C05493=1117.281,-65.338,-48.036,179.657,5.180,148.998
C05494=1117.275,-65.089,-48.047,179.658,5.185,148.999
C05495=1117.270,-64.839,-48.058,179.658,5.190,149.000
C05496=1117.264,-64.590,-48.069,179.659,5.196,149.001
C05497=1117.259,-64.339,-48.080,179.659,5.201,149.001
C05498=1117.254,-64.090,-48.090,179.659,5.206,149.003
C05499=1117.249,-63.840,-48.101,179.660,5.211,149.004
C05500=1117.244,-63.590,-48.112,179.660,5.216,149.004
C05501=1117.239,-63.341,-48.123,179.661,5.222,149.005
C05502=1117.233,-63.091,-48.134,179.661,5.227,149.007
C05503=1117.228,-62.842,-48.145,179.661,5.231,149.007
C05504=1117.223,-62.592,-48.156,179.662,5.237,149.008
C05505=1117.217,-62.342,-48.166,179.663,5.242,149.009
C05506=1117.212,-62.093,-48.178,179.664,5.247,149.010
C05507=1117.207,-61.842,-48.189,179.664,5.252,149.011
C05508=1117.202,-61.593,-48.200,179.665,5.258,149.012
C05509=1117.197,-61.343,-48.210,179.665,5.263,149.013
C05510=1117.191,-61.093,-48.222,179.665,5.268,149.014
C05511=1117.186,-60.844,-48.233,179.666,5.273,149.015
C05512=1117.181,-60.594,-48.244,179.667,5.278,149.016
C05513=1117.176,-60.344,-48.255,179.668,5.283,149.017
C05514=1117.170,-60.094,-48.266,179.668,5.288,149.018
C05515=1117.166,-59.880,-48.276,179.668,5.292,149.019
C05516=1117.161,-59.664,-48.285,179.668,5.296,149.020
C05517=1117.157,-59.450,-48.294,179.668,5.301,149.021
C05518=1117.153,-59.235,-48.304,179.668,5.305,149.022
C05519=1117.148,-59.020,-48.313,179.668,5.309,149.022
C05520=1117.143,-58.805,-48.323,179.668,5.313,149.023
C05521=1117.139,-58.590,-48.333,179.667,5.317,149.024
C05522=1117.134,-58.375,-48.343,179.667,5.321,149.025
C05523=1117.129,-58.124,-48.353,179.668,5.325,149.026
C05524=1117.123,-57.875,-48.365,179.667,5.330,149.027
C05525=1117.119,-57.626,-48.376,179.667,5.335,149.028
C05526=1117.114,-57.376,-48.387,179.667,5.339,149.029
C05527=1117.108,-57.126,-48.398,179.666,5.344,149.031
C05528=1117.103,-56.877,-48.409,179.666,5.349,149.032
C05529=1117.098,-56.627,-48.421,179.666,5.353,149.033
C05530=1117.093,-56.377,-48.433,179.666,5.358,149.034
C05531=1117.087,-56.127,-48.443,179.666,5.362,149.035
C05532=1117.082,-55.877,-48.455,179.666,5.367,149.036
C05533=1117.077,-55.628,-48.466,179.666,5.372,149.037
C05534=1117.072,-55.379,-48.477,179.666,5.376,149.038
C05535=1117.066,-55.128,-48.488,179.665,5.381,149.039
C05536=1117.061,-54.879,-48.499,179.665,5.386,149.040
C05537=1117.056,-54.629,-48.511,179.665,5.391,149.041
C05538=1117.051,-54.380,-48.522,179.665,5.396,149.042
C05539=1117.046,-54.130,-48.533,179.664,5.400,149.043
C05540=1117.040,-53.880,-48.545,179.665,5.405,149.044
C05541=1117.036,-53.630,-48.556,179.664,5.409,149.045
C05542=1117.029,-53.381,-48.567,179.664,5.414,149.047
C05543=1117.025,-53.131,-48.579,179.664,5.419,149.048
C05544=1117.019,-52.881,-48.591,179.664,5.423,149.049
C05545=1117.015,-52.632,-48.602,179.664,5.429,149.050
C05546=1117.009,-52.382,-48.613,179.663,5.432,149.051
C05547=1117.004,-52.132,-48.624,179.663,5.438,149.052
C05548=1116.998,-51.882,-48.636,179.663,5.443,149.053
C05549=1116.994,-51.633,-48.647,179.663,5.447,149.054
C05550=1116.987,-51.383,-48.659,179.663,5.452,149.055
C05551=1116.983,-51.134,-48.670,179.662,5.456,149.056
C05552=1116.977,-50.884,-48.682,179.663,5.461,149.057
C05553=1116.973,-50.634,-48.693,179.663,5.466,149.058
C05554=1116.967,-50.384,-48.705,179.662,5.470,149.060
C05555=1116.962,-50.135,-48.716,179.662,5.476,149.061
C05556=1116.957,-49.885,-48.728,179.662,5.479,149.062
C05557=1116.952,-49.636,-48.739,179.662,5.485,149.063
C05558=1116.946,-49.385,-48.750,179.662,5.490,149.064
C05559=1116.941,-49.136,-48.762,179.661,5.494,149.065
C05560=1116.935,-48.886,-48.773,179.661,5.499,149.066
C05561=1116.931,-48.637,-48.784,179.661,5.503,149.067
C05562=1116.925,-48.387,-48.796,179.661,5.508,149.068
C05563=1116.920,-48.137,-48.808,179.661,5.513,149.069
C05564=1116.915,-47.887,-48.819,179.660,5.517,149.070
C05565=1116.909,-47.638,-48.831,179.660,5.522,149.071
C05566=1116.904,-47.388,-48.842,179.660,5.526,149.072
C05567=1116.899,-47.138,-48.854,179.660,5.532,149.073
C05568=1116.894,-46.889,-48.865,179.660,5.537,149.075
C05569=1116.889,-46.639,-48.877,179.659,5.541,149.076
C05570=1116.884,-46.390,-48.890,179.660,5.546,149.077
C05571=1116.879,-46.174,-48.899,179.660,5.550,149.078
C05572=1116.875,-45.959,-48.909,179.659,5.554,149.079
C05573=1116.870,-45.744,-48.919,179.659,5.558,149.079
C05574=1116.866,-45.529,-48.929,179.659,5.562,149.081
C05575=1116.862,-45.315,-48.939,179.658,5.566,149.081
C05576=1116.857,-45.099,-48.950,179.658,5.570,149.082
C05577=1116.852,-44.885,-48.959,179.659,5.575,149.083
C05578=1116.847,-44.670,-48.969,179.658,5.579,149.084
C05579=1116.843,-44.421,-48.981,179.658,5.583,149.085
C05580=1116.837,-44.171,-48.993,179.658,5.588,149.086
C05581=1116.832,-43.921,-49.005,179.658,5.592,149.087
C05582=1116.827,-43.671,-49.016,179.658,5.597,149.089
C05583=1116.822,-43.422,-49.028,179.658,5.602,149.089
C05584=1116.817,-43.172,-49.040,179.657,5.606,149.091
C05585=1116.812,-42.922,-49.052,179.657,5.611,149.092
C05586=1116.806,-42.672,-49.063,179.658,5.617,149.093
C05587=1116.801,-42.422,-49.075,179.660,5.622,149.093
C05588=1116.796,-42.174,-49.086,179.661,5.628,149.094
C05589=1116.791,-41.924,-49.099,179.662,5.633,149.095
C05590=1116.785,-41.674,-49.111,179.663,5.638,149.096
C05591=1116.780,-41.424,-49.123,179.664,5.644,149.097
C05592=1116.775,-41.175,-49.134,179.665,5.649,149.098
C05593=1116.770,-40.925,-49.147,179.666,5.654,149.098
C05594=1116.765,-40.676,-49.158,179.667,5.659,149.099
C05595=1116.759,-40.426,-49.170,179.668,5.665,149.100
C05596=1116.754,-40.176,-49.182,179.669,5.669,149.101
C05597=1116.749,-39.927,-49.194,179.670,5.675,149.102
C05598=1116.744,-39.677,-49.206,179.672,5.680,149.103
C05599=1116.738,-39.427,-49.218,179.672,5.685,149.103
C05600=1116.733,-39.177,-49.231,179.673,5.690,149.104
C05601=1116.729,-38.928,-49.242,179.674,5.695,149.105
C05602=1116.723,-38.678,-49.254,179.675,5.699,149.106
C05603=1116.718,-38.429,-49.266,179.676,5.705,149.107
C05604=1116.713,-38.179,-49.278,179.676,5.710,149.108
C05605=1116.707,-37.929,-49.290,179.677,5.714,149.108
C05606=1116.702,-37.679,-49.303,179.678,5.719,149.109
C05607=1116.697,-37.430,-49.314,179.679,5.724,149.110
C05608=1116.692,-37.180,-49.327,179.680,5.729,149.111
C05609=1116.687,-36.930,-49.339,179.680,5.733,149.112
C05610=1116.681,-36.681,-49.350,179.681,5.738,149.113
C05611=1116.676,-36.431,-49.363,179.682,5.743,149.113
C05612=1116.671,-36.181,-49.375,179.683,5.748,149.114
C05613=1116.666,-35.932,-49.387,179.683,5.753,149.115
C05614=1116.660,-35.682,-49.399,179.683,5.757,149.116
C05615=1116.655,-35.433,-49.412,179.684,5.762,149.117
C05616=1116.650,-35.183,-49.423,179.685,5.766,149.117
C05617=1116.645,-34.934,-49.436,179.685,5.771,149.118
C05618=1116.640,-34.684,-49.448,179.685,5.775,149.119
C05619=1116.635,-34.435,-49.460,179.686,5.780,149.120
C05620=1116.629,-34.185,-49.472,179.687,5.784,149.121
C05621=1116.625,-33.935,-49.485,179.687,5.789,149.122
C05622=1116.619,-33.685,-49.497,179.687,5.794,149.123
C05623=1116.614,-33.435,-49.510,179.687,5.798,149.124
C05624=1116.609,-33.186,-49.522,179.688,5.802,149.124
C05625=1116.604,-32.936,-49.534,179.689,5.807,149.125
C05626=1116.599,-32.687,-49.547,179.689,5.811,149.126
C05627=1116.594,-32.472,-49.557,179.689,5.815,149.127
C05628=1116.589,-32.257,-49.568,179.689,5.819,149.128
C05629=1116.586,-32.042,-49.578,179.690,5.823,149.128
C05630=1116.581,-31.827,-49.589,179.690,5.826,149.129
C05631=1116.577,-31.612,-49.600,179.690,5.830,149.130
C05632=1116.572,-31.397,-49.610,179.690,5.834,149.131
C05633=1116.568,-31.183,-49.621,179.690,5.838,149.132
C05634=1116.562,-30.968,-49.632,179.690,5.841,149.132
C05635=1116.557,-30.718,-49.644,179.690,5.845,149.133
C05636=1116.553,-30.468,-49.657,179.690,5.850,149.134
C05637=1116.547,-30.218,-49.669,179.690,5.854,149.135
C05638=1116.542,-29.969,-49.682,179.690,5.858,149.136
C05639=1116.537,-29.720,-49.694,179.690,5.863,149.137
C05640=1116.532,-29.470,-49.706,179.690,5.867,149.138
C05641=1116.527,-29.221,-49.719,179.690,5.871,149.139
C05642=1116.522,-28.971,-49.732,179.690,5.876,149.140
C05643=1116.517,-28.721,-49.744,179.690,5.880,149.141
C05644=1116.512,-28.471,-49.756,179.689,5.884,149.142
C05645=1116.506,-28.222,-49.769,179.689,5.888,149.143
C05646=1116.501,-27.972,-49.781,179.689,5.892,149.144
C05647=1116.496,-27.723,-49.793,179.689,5.896,149.145
C05648=1116.491,-27.473,-49.806,179.689,5.901,149.146
C05649=1116.486,-27.223,-49.819,179.688,5.906,149.147
C05650=1116.480,-26.973,-49.831,179.688,5.910,149.148
C05651=1116.475,-26.724,-49.844,179.687,5.914,149.149
C05652=1116.470,-26.475,-49.857,179.687,5.918,149.150
C05653=1116.465,-26.224,-49.870,179.686,5.922,149.151
C05654=1116.460,-25.975,-49.881,179.686,5.927,149.152
C05655=1116.455,-25.725,-49.894,179.686,5.930,149.153
C05656=1116.450,-25.476,-49.907,179.686,5.936,149.154
C05657=1116.444,-25.227,-49.919,179.687,5.941,149.155
C05658=1116.440,-24.977,-49.932,179.687,5.946,149.156
C05659=1116.434,-24.726,-49.945,179.688,5.951,149.157
C05660=1116.429,-24.477,-49.957,179.688,5.955,149.158
C05661=1116.424,-24.228,-49.970,179.689,5.960,149.159
C05662=1116.418,-23.978,-49.983,179.689,5.965,149.160
C05663=1116.414,-23.728,-49.996,179.690,5.969,149.160
C05664=1116.409,-23.479,-50.008,179.691,5.974,149.161
C05665=1116.403,-23.229,-50.021,179.692,5.979,149.162
C05666=1116.397,-22.979,-50.033,179.692,5.984,149.163
C05667=1116.393,-22.729,-50.046,179.693,5.989,149.164
C05668=1116.388,-22.480,-50.059,179.693,5.994,149.165
C05669=1116.383,-22.231,-50.071,179.694,5.998,149.166
C05670=1116.377,-21.981,-50.085,179.694,6.003,149.167
C05671=1116.372,-21.731,-50.098,179.694,6.008,149.168
C05672=1116.367,-21.482,-50.110,179.695,6.013,149.169
C05673=1116.362,-21.233,-50.123,179.695,6.017,149.169
C05674=1116.357,-20.982,-50.136,179.696,6.022,149.170
C05675=1116.352,-20.733,-50.149,179.696,6.027,149.171
C05676=1116.347,-20.484,-50.161,179.697,6.031,149.172
C05677=1116.341,-20.234,-50.174,179.698,6.036,149.173
C05678=1116.336,-19.984,-50.188,179.698,6.041,149.174
C05679=1116.331,-19.735,-50.200,179.699,6.045,149.175
C05680=1116.326,-19.485,-50.213,179.699,6.050,149.175
C05681=1116.321,-19.235,-50.226,179.700,6.055,149.176
C05682=1116.316,-18.986,-50.239,179.701,6.060,149.177
C05683=1116.311,-18.771,-50.250,179.701,6.064,149.178
C05684=1116.307,-18.556,-50.261,179.702,6.067,149.179
C05685=1116.302,-18.341,-50.272,179.702,6.072,149.179
C05686=1116.297,-18.126,-50.283,179.702,6.076,149.180
C05687=1116.293,-17.912,-50.294,179.703,6.080,149.181
C05688=1116.289,-17.697,-50.306,179.704,6.084,149.181
C05689=1116.284,-17.482,-50.317,179.704,6.088,149.182
C05690=1116.280,-17.268,-50.328,179.705,6.092,149.183
C05691=1116.275,-17.018,-50.341,179.705,6.097,149.184
C05692=1116.270,-16.768,-50.354,179.706,6.101,149.185
C05693=1116.265,-16.518,-50.367,179.707,6.106,149.186
C05694=1116.260,-16.269,-50.380,179.707,6.110,149.186
C05695=1116.254,-16.020,-50.394,179.708,6.115,149.187
C05696=1116.250,-15.770,-50.407,179.708,6.120,149.188
C05697=1116.244,-15.520,-50.420,179.709,6.124,149.189
C05698=1116.239,-15.271,-50.433,179.710,6.129,149.190
C05699=1116.234,-15.021,-50.446,179.710,6.134,149.191
C05700=1116.228,-14.771,-50.459,179.711,6.138,149.192
C05701=1116.224,-14.522,-50.473,179.711,6.143,149.192
C05702=1116.219,-14.272,-50.485,179.712,6.147,149.193
C05703=1116.213,-14.023,-50.498,179.713,6.152,149.194
C05704=1116.209,-13.773,-50.511,179.713,6.157,149.195
C05705=1116.203,-13.524,-50.525,179.714,6.162,149.196
C05706=1116.198,-13.274,-50.538,179.715,6.166,149.196
C05707=1116.193,-13.024,-50.551,179.715,6.171,149.197
C05708=1116.188,-12.774,-50.564,179.716,6.175,149.198
C05709=1116.183,-12.525,-50.578,179.716,6.180,149.199
C05710=1116.178,-12.275,-50.591,179.717,6.184,149.200
C05711=1116.172,-12.025,-50.604,179.718,6.189,149.201
C05712=1116.167,-11.777,-50.618,179.718,6.194,149.202
C05713=1116.162,-11.526,-50.631,179.719,6.199,149.202
C05714=1116.157,-11.277,-50.644,179.719,6.202,149.203
C05715=1116.152,-11.027,-50.658,179.719,6.207,149.204
C05716=1116.147,-10.778,-50.671,179.720,6.212,149.205
C05717=1116.142,-10.528,-50.684,179.721,6.216,149.206
C05718=1116.137,-10.279,-50.698,179.721,6.221,149.206
C05719=1116.131,-10.029,-50.711,179.722,6.225,149.207
C05720=1116.127,-9.780,-50.725,179.722,6.230,149.208
C05721=1116.121,-9.530,-50.738,179.723,6.234,149.209
C05722=1116.116,-9.280,-50.751,179.724,6.239,149.210
C05723=1116.111,-9.031,-50.765,179.724,6.244,149.211
C05724=1116.106,-8.781,-50.778,179.725,6.248,149.211
C05725=1116.101,-8.532,-50.792,179.726,6.253,149.212
C05726=1116.095,-8.282,-50.805,179.726,6.258,149.213
C05727=1116.091,-8.033,-50.819,179.727,6.262,149.214
C05728=1116.085,-7.783,-50.832,179.727,6.266,149.215
C05729=1116.081,-7.534,-50.846,179.728,6.271,149.216
C05730=1116.075,-7.284,-50.859,179.728,6.275,149.216
C05731=1116.070,-7.034,-50.873,179.729,6.280,149.217
C05732=1116.066,-6.784,-50.886,179.730,6.284,149.218
C05733=1116.060,-6.535,-50.900,179.730,6.289,149.219
C05734=1116.055,-6.285,-50.914,179.731,6.293,149.220
C05735=1116.050,-6.036,-50.927,179.732,6.298,149.220
C05736=1116.045,-5.786,-50.940,179.732,6.303,149.221
C05737=1116.039,-5.537,-50.954,179.733,6.308,149.222
C05738=1116.035,-5.287,-50.967,179.733,6.311,149.223
C05739=1116.030,-5.073,-50.979,179.734,6.316,149.224
C05740=1116.026,-4.858,-50.991,179.734,6.319,149.224
C05741=1116.021,-4.643,-51.002,179.735,6.324,149.225
C05742=1116.018,-4.428,-51.015,179.736,6.327,149.226
C05743=1116.013,-4.214,-51.026,179.736,6.331,149.226
C05744=1116.009,-3.999,-51.038,179.737,6.335,149.227
C05745=1116.004,-3.785,-51.050,179.737,6.339,149.228
C05746=1116.000,-3.569,-51.061,179.737,6.343,149.229
C05747=1115.994,-3.320,-51.075,179.738,6.347,149.229
C05748=1115.989,-3.070,-51.089,179.739,6.352,149.230
C05749=1115.984,-2.820,-51.103,179.739,6.356,149.231
C05750=1115.979,-2.572,-51.117,179.740,6.361,149.232
C05751=1115.974,-2.321,-51.130,179.741,6.365,149.233
C05752=1115.969,-2.072,-51.144,179.741,6.370,149.234
C05753=1115.964,-1.823,-51.158,179.742,6.375,149.234
C05754=1115.959,-1.573,-51.171,179.742,6.378,149.235
C05755=1115.954,-1.324,-51.185,179.743,6.383,149.236
C05756=1115.949,-1.074,-51.199,179.743,6.388,149.237
C05757=1115.944,-0.824,-51.214,179.744,6.393,149.238
C05758=1115.938,-0.575,-51.226,179.745,6.397,149.238
C05759=1115.934,-0.325,-51.241,179.745,6.402,149.239
C05760=1115.929,-0.075,-51.255,179.746,6.406,149.240
C05761=1115.923,0.174,-51.269,179.747,6.411,149.241
C05762=1115.918,0.424,-51.282,179.747,6.415,149.242
C05763=1115.913,0.674,-51.297,179.747,6.419,149.243
C05764=1115.908,0.922,-51.310,179.748,6.424,149.244
C05765=1115.903,1.172,-51.324,179.749,6.428,149.244
C05766=1115.898,1.422,-51.338,179.749,6.433,149.245
C05767=1115.892,1.671,-51.352,179.750,6.438,149.246
C05768=1115.887,1.921,-51.366,179.751,6.443,149.247
C05769=1115.882,2.171,-51.380,179.752,6.447,149.248
C05770=1115.878,2.420,-51.394,179.752,6.452,149.248
C05771=1115.873,2.669,-51.408,179.752,6.456,149.249
C05772=1115.868,2.919,-51.422,179.753,6.460,149.250
C05773=1115.863,3.169,-51.436,179.754,6.465,149.251
C05774=1115.857,3.418,-51.450,179.754,6.469,149.252
C05775=1115.852,3.668,-51.464,179.755,6.474,149.253
C05776=1115.847,3.918,-51.478,179.755,6.479,149.254
C05777=1115.842,4.167,-51.492,179.756,6.483,149.254
C05778=1115.836,4.416,-51.506,179.757,6.488,149.255
C05779=1115.831,4.666,-51.521,179.757,6.492,149.256
C05780=1115.826,4.916,-51.535,179.757,6.496,149.257
C05781=1115.822,5.165,-51.549,179.758,6.501,149.258
C05782=1115.817,5.414,-51.562,179.758,6.506,149.259
C05783=1115.812,5.664,-51.577,179.759,6.510,149.259
C05784=1115.807,5.914,-51.591,179.760,6.515,149.260
C05785=1115.802,6.163,-51.605,179.760,6.520,149.261
C05786=1115.797,6.413,-51.620,179.761,6.524,149.262
C05787=1115.791,6.662,-51.634,179.761,6.529,149.263
C05788=1115.786,6.912,-51.648,179.762,6.534,149.264
C05789=1115.781,7.161,-51.662,179.762,6.537,149.264
C05790=1115.776,7.411,-51.676,179.763,6.542,149.265
C05791=1115.771,7.660,-51.690,179.763,6.547,149.266
C05792=1115.766,7.910,-51.705,179.764,6.551,149.267
C05793=1115.761,8.160,-51.719,179.765,6.556,149.268
C05794=1115.756,8.409,-51.733,179.765,6.561,149.269
C05795=1115.750,8.699,-51.750,179.766,6.566,149.270
C05796=1115.744,8.990,-51.767,179.766,6.571,149.271
C05797=1115.737,9.281,-51.783,179.767,6.577,149.272
C05798=1115.732,9.572,-51.800,179.768,6.582,149.273
C05799=1115.727,9.822,-51.815,179.769,6.586,149.273
C05800=1115.722,10.072,-51.829,179.769,6.591,149.274
C05801=1115.717,10.320,-51.844,179.770,6.596,149.275
C05802=1115.712,10.570,-51.858,179.770,6.600,149.276
C05803=1115.707,10.819,-51.872,179.771,6.605,149.277
C05804=1115.702,11.069,-51.886,179.772,6.610,149.278
C05805=1115.697,11.319,-51.901,179.772,6.614,149.278
C05806=1115.692,11.568,-51.916,179.773,6.619,149.279
C05807=1115.687,11.818,-51.931,179.774,6.623,149.280
C05808=1115.681,12.067,-51.944,179.774,6.628,149.281
C05809=1115.676,12.317,-51.959,179.775,6.633,149.282
C05810=1115.671,12.566,-51.973,179.776,6.637,149.282
C05811=1115.667,12.816,-51.988,179.777,6.642,149.283
C05812=1115.662,13.065,-52.002,179.777,6.646,149.284
C05813=1115.657,13.315,-52.017,179.778,6.650,149.285
C05814=1115.651,13.564,-52.032,179.778,6.655,149.286
C05815=1115.646,13.814,-52.046,179.779,6.659,149.287
C05816=1115.641,14.064,-52.061,179.780,6.664,149.287
C05817=1115.636,14.313,-52.075,179.780,6.668,149.288
C05818=1115.632,14.563,-52.090,179.781,6.673,149.289
C05819=1115.625,14.812,-52.104,179.782,6.677,149.290
C05820=1115.620,15.062,-52.119,179.782,6.682,149.291
C05821=1115.616,15.311,-52.134,179.783,6.686,149.291
C05822=1115.611,15.560,-52.148,179.784,6.691,149.292
C05823=1115.606,15.810,-52.162,179.785,6.695,149.293
C05824=1115.600,16.060,-52.178,179.786,6.700,149.294
C05825=1115.596,16.309,-52.192,179.786,6.705,149.295
C05826=1115.591,16.558,-52.207,179.787,6.708,149.295
C05827=1115.586,16.808,-52.221,179.787,6.713,149.296
C05828=1115.580,17.058,-52.236,179.788,6.717,149.297
C05829=1115.576,17.307,-52.251,179.789,6.722,149.298
C05830=1115.571,17.557,-52.266,179.790,6.726,149.298
C05831=1115.563,17.945,-52.289,179.791,6.734,149.300
C05832=1115.555,18.333,-52.312,179.792,6.740,149.301
C05833=1115.547,18.721,-52.335,179.793,6.747,149.302
C05834=1115.540,19.109,-52.358,179.794,6.754,149.303
C05835=1115.535,19.358,-52.373,179.795,6.758,149.304
C05836=1115.529,19.608,-52.388,179.796,6.763,149.305
C05837=1115.524,19.858,-52.402,179.797,6.767,149.305
C05838=1115.520,20.107,-52.417,179.797,6.772,149.306
C05839=1115.514,20.357,-52.432,179.798,6.776,149.307
C05840=1115.509,20.606,-52.447,179.799,6.781,149.307
C05841=1115.504,20.856,-52.462,179.800,6.785,149.308
C05842=1115.499,21.105,-52.477,179.801,6.790,149.309
C05843=1115.494,21.354,-52.492,179.801,6.794,149.310
C05844=1115.489,21.604,-52.507,179.802,6.798,149.311
C05845=1115.484,21.853,-52.522,179.803,6.802,149.311
C05846=1115.478,22.103,-52.537,179.804,6.807,149.312
C05847=1115.475,22.317,-52.550,179.804,6.810,149.313
C05848=1115.470,22.532,-52.563,179.805,6.815,149.313
C05849=1115.466,22.746,-52.575,179.806,6.818,149.314
C05850=1115.461,22.960,-52.589,179.807,6.822,149.314
C05851=1115.458,23.175,-52.601,179.808,6.826,149.315
C05852=1115.453,23.390,-52.614,179.808,6.829,149.316
C05853=1115.449,23.604,-52.628,179.809,6.834,149.316
C05854=1115.445,23.819,-52.640,179.809,6.837,149.317
C05855=1115.439,24.068,-52.656,179.810,6.841,149.318
C05856=1115.434,24.318,-52.670,179.812,6.846,149.318
C05857=1115.429,24.567,-52.686,179.812,6.850,149.319
C05858=1115.424,24.816,-52.701,179.813,6.854,149.320
C05859=1115.419,25.067,-52.715,179.814,6.858,149.321
C05860=1115.414,25.316,-52.730,179.815,6.863,149.321
C05861=1115.409,25.565,-52.746,179.815,6.867,149.322
C05862=1115.405,25.815,-52.761,179.816,6.872,149.323
C05863=1115.399,26.065,-52.776,179.817,6.876,149.323
C05864=1115.394,26.314,-52.791,179.818,6.880,149.324
C05865=1115.389,26.563,-52.807,179.819,6.885,149.325
C05866=1115.384,26.812,-52.822,179.819,6.888,149.326
C05867=1115.379,27.062,-52.837,179.820,6.893,149.326
C05868=1115.374,27.312,-52.852,179.821,6.897,149.327
C05869=1115.369,27.562,-52.868,179.823,6.901,149.328
C05870=1115.365,27.811,-52.883,179.824,6.906,149.328
C05871=1115.359,28.060,-52.898,179.824,6.910,149.329
C05872=1115.354,28.310,-52.914,179.825,6.915,149.330
C05873=1115.349,28.559,-52.929,179.826,6.918,149.330
C05874=1115.344,28.808,-52.944,179.827,6.923,149.331
C05875=1115.339,29.058,-52.959,179.828,6.927,149.332
C05876=1115.334,29.308,-52.975,179.829,6.931,149.332
C05877=1115.329,29.557,-52.990,179.829,6.936,149.333
C05878=1115.324,29.806,-53.005,179.830,6.940,149.334
C05879=1115.319,30.056,-53.021,179.832,6.945,149.335
C05880=1115.315,30.306,-53.036,179.833,6.949,149.335
C05881=1115.309,30.555,-53.052,179.833,6.952,149.336
C05882=1115.304,30.804,-53.067,179.834,6.957,149.337
C05883=1115.299,31.053,-53.082,179.835,6.961,149.337
C05884=1115.294,31.304,-53.098,179.836,6.965,149.338
C05885=1115.289,31.553,-53.114,179.837,6.970,149.338
C05886=1115.284,31.802,-53.129,179.838,6.974,149.339
C05887=1115.279,32.051,-53.144,179.839,6.978,149.340
C05888=1115.274,32.302,-53.160,179.840,6.982,149.340
C05889=1115.269,32.551,-53.175,179.840,6.986,149.341
C05890=1115.264,32.800,-53.191,179.842,6.991,149.342
C05891=1115.259,33.049,-53.207,179.843,6.995,149.343
C05892=1115.254,33.300,-53.223,179.844,6.999,149.343
C05893=1115.249,33.549,-53.238,179.845,7.004,149.344
C05894=1115.244,33.798,-53.253,179.846,7.008,149.345
C05895=1115.238,34.047,-53.269,179.846,7.011,149.345
C05896=1115.234,34.297,-53.284,179.847,7.016,149.346
C05897=1115.229,34.546,-53.300,179.848,7.020,149.347
C05898=1115.224,34.795,-53.316,179.849,7.024,149.347
C05899=1115.219,35.046,-53.332,179.850,7.029,149.348
C05900=1115.215,35.295,-53.347,179.852,7.033,149.348
C05901=1115.209,35.544,-53.363,179.853,7.037,149.349
C05902=1115.204,35.794,-53.378,179.854,7.040,149.350
C05903=1115.200,36.008,-53.392,179.855,7.045,149.350
C05904=1115.195,36.222,-53.406,179.855,7.048,149.351
C05905=1115.191,36.436,-53.419,179.856,7.051,149.351
C05906=1115.186,36.651,-53.432,179.857,7.056,149.352
C05907=1115.182,36.866,-53.446,179.858,7.059,149.352
C05908=1115.178,37.080,-53.460,179.858,7.062,149.353
C05909=1115.174,37.294,-53.473,179.860,7.066,149.353
C05910=1115.170,37.509,-53.487,179.860,7.070,149.354
C05911=1115.165,37.758,-53.502,179.861,7.074,149.355
C05912=1115.160,38.008,-53.518,179.863,7.078,149.355
C05913=1115.155,38.258,-53.534,179.863,7.082,149.356
C05914=1115.150,38.507,-53.550,179.864,7.086,149.357
C05915=1115.144,38.756,-53.566,179.866,7.090,149.357
C05916=1115.140,39.006,-53.582,179.867,7.095,149.358
C05917=1115.135,39.255,-53.597,179.868,7.099,149.358
C05918=1115.130,39.504,-53.613,179.869,7.103,149.359
C05919=1115.125,39.754,-53.629,179.870,7.107,149.360
C05920=1115.120,40.004,-53.645,179.871,7.111,149.360
C05921=1115.115,40.253,-53.661,179.872,7.115,149.361
C05922=1115.110,40.502,-53.677,179.873,7.119,149.362
C05923=1115.105,40.751,-53.693,179.874,7.123,149.362
C05924=1115.100,41.001,-53.709,179.875,7.128,149.363
C05925=1115.095,41.251,-53.725,179.876,7.132,149.363
C05926=1115.090,41.500,-53.741,179.878,7.136,149.364
C05927=1115.085,41.750,-53.757,179.878,7.140,149.365
C05928=1115.079,41.999,-53.773,179.879,7.144,149.365
C05929=1115.075,42.249,-53.789,179.880,7.148,149.366
C05930=1115.069,42.498,-53.805,179.881,7.152,149.367
C05931=1115.066,42.747,-53.821,179.883,7.156,149.367
C05932=1115.060,42.997,-53.836,179.884,7.161,149.368
C05933=1115.056,43.246,-53.853,179.884,7.164,149.368
C05934=1115.050,43.495,-53.869,179.886,7.168,149.369
C05935=1115.046,43.745,-53.885,179.887,7.172,149.369
C05936=1115.041,43.994,-53.901,179.888,7.177,149.370
C05937=1115.036,44.244,-53.918,179.889,7.181,149.371
C05938=1115.030,44.493,-53.934,179.890,7.185,149.371
C05939=1115.026,44.743,-53.951,179.892,7.189,149.372
C05940=1115.020,44.992,-53.966,179.892,7.193,149.372
C05941=1115.016,45.242,-53.983,179.893,7.197,149.373
C05942=1115.010,45.491,-53.998,179.894,7.201,149.374
C05943=1115.006,45.741,-54.015,179.896,7.205,149.374
C05944=1115.000,45.990,-54.031,179.897,7.210,149.375
C05945=1114.996,46.240,-54.047,179.898,7.214,149.375
C05946=1114.991,46.488,-54.064,179.899,7.217,149.376
C05947=1114.986,46.739,-54.080,179.900,7.221,149.376
C05948=1114.981,46.987,-54.096,179.901,7.226,149.377
C05949=1114.976,47.237,-54.112,179.902,7.230,149.378
C05950=1114.971,47.486,-54.128,179.904,7.234,149.378
C05951=1114.967,47.736,-54.145,179.905,7.238,149.379
C05952=1114.960,47.985,-54.161,179.906,7.242,149.380
C05953=1114.956,48.235,-54.178,179.907,7.246,149.380
C05954=1114.951,48.484,-54.194,179.908,7.250,149.381
C05955=1114.946,48.734,-54.210,179.909,7.254,149.381
C05956=1114.942,48.983,-54.227,179.911,7.258,149.382
C05957=1114.937,49.232,-54.243,179.912,7.262,149.382
C05958=1114.932,49.482,-54.259,179.913,7.266,149.383
C05959=1114.927,49.696,-54.274,179.914,7.270,149.383
C05960=1114.923,49.910,-54.288,179.915,7.273,149.384
C05961=1114.918,50.125,-54.301,179.916,7.277,149.384
C05962=1114.914,50.339,-54.316,179.917,7.280,149.385
C05963=1114.911,50.554,-54.330,179.918,7.283,149.385
C05964=1114.906,50.768,-54.344,179.919,7.287,149.386
C05965=1114.902,50.982,-54.358,179.920,7.290,149.386
C05966=1114.897,51.196,-54.372,179.921,7.294,149.387
C05967=1114.893,51.446,-54.389,179.922,7.298,149.387
C05968=1114.887,51.695,-54.406,179.923,7.302,149.388
C05969=1114.883,51.944,-54.422,179.925,7.306,149.388
C05970=1114.878,52.194,-54.438,179.926,7.310,149.389
C05971=1114.873,52.443,-54.455,179.927,7.314,149.389
C05972=1114.868,52.693,-54.472,179.928,7.318,149.390
C05973=1114.863,52.942,-54.489,179.929,7.322,149.391
C05974=1114.858,53.191,-54.505,179.931,7.326,149.391
C05975=1114.854,53.441,-54.522,179.932,7.330,149.392
C05976=1114.847,53.690,-54.538,179.933,7.334,149.392
C05977=1114.843,53.940,-54.554,179.934,7.339,149.393
C05978=1114.838,54.189,-54.571,179.935,7.342,149.393
C05979=1114.833,54.438,-54.588,179.936,7.346,149.394
C05980=1114.828,54.688,-54.605,179.938,7.350,149.394
C05981=1114.824,54.937,-54.621,179.939,7.354,149.395
C05982=1114.818,55.187,-54.638,179.941,7.358,149.396
C05983=1114.813,55.436,-54.655,179.942,7.362,149.396
C05984=1114.809,55.686,-54.672,179.943,7.366,149.397
C05985=1114.803,55.935,-54.688,179.944,7.370,149.397
C05986=1114.799,56.184,-54.705,179.945,7.374,149.398
C05987=1114.794,56.434,-54.722,179.946,7.378,149.398
C05988=1114.789,56.683,-54.739,179.947,7.382,149.399
C05989=1114.784,56.932,-54.755,179.949,7.386,149.399
C05990=1114.779,57.182,-54.773,179.950,7.391,149.400
C05991=1114.774,57.431,-54.789,179.952,7.394,149.401
C05992=1114.769,57.680,-54.806,179.952,7.398,149.401
C05993=1114.764,57.930,-54.823,179.954,7.402,149.402
C05994=1114.759,58.179,-54.840,179.955,7.406,149.402
C05995=1114.754,58.429,-54.857,179.956,7.410,149.403
C05996=1114.749,58.678,-54.873,179.958,7.414,149.403
C05997=1114.744,58.927,-54.891,179.959,7.418,149.404
C05998=1114.740,59.177,-54.908,179.961,7.422,149.404
C05999=1114.735,59.426,-54.924,179.961,7.426,149.405
C06000=1114.729,59.675,-54.941,179.963,7.430,149.405
C06001=1114.725,59.925,-54.958,179.964,7.434,149.406
C06002=1114.720,60.175,-54.975,179.965,7.438,149.406
C06003=1114.715,60.424,-54.992,179.966,7.442,149.407
C06004=1114.710,60.673,-55.010,179.968,7.446,149.407
C06005=1114.705,60.922,-55.026,179.969,7.450,149.408
C06006=1114.700,61.172,-55.043,179.971,7.454,149.409
C06007=1114.696,61.421,-55.060,179.972,7.457,149.409
C06008=1114.690,61.671,-55.077,179.973,7.462,149.410
C06009=1114.686,61.920,-55.095,179.974,7.466,149.410
C06010=1114.680,62.169,-55.112,179.975,7.470,149.411
C06011=1114.676,62.419,-55.128,179.977,7.474,149.411
C06012=1114.671,62.668,-55.146,179.978,7.478,149.412
C06013=1114.666,62.918,-55.164,179.980,7.482,149.412
C06014=1114.661,63.167,-55.180,179.981,7.486,149.413
C06015=1114.656,63.381,-55.195,179.982,7.489,149.413
C06016=1114.652,63.595,-55.210,179.983,7.492,149.413
C06017=1114.648,63.809,-55.225,179.985,7.496,149.414
C06018=1114.644,64.024,-55.239,179.985,7.499,149.414
C06019=1114.640,64.238,-55.254,179.986,7.503,149.415
C06020=1114.636,64.452,-55.269,179.988,7.506,149.415
C06021=1114.631,64.666,-55.284,179.988,7.510,149.416
C06022=1114.628,64.881,-55.298,179.989,7.513,149.416
C06023=1114.623,65.130,-55.316,179.991,7.517,149.417
C06024=1114.618,65.380,-55.334,179.993,7.521,149.417
C06025=1114.613,65.628,-55.350,179.994,7.525,149.418
C06026=1114.607,65.878,-55.367,179.995,7.529,149.418
C06027=1114.603,66.127,-55.385,179.997,7.533,149.419
C06028=1114.598,66.377,-55.402,179.998,7.537,149.419
C06029=1114.593,66.626,-55.420,179.999,7.540,149.420
C06030=1114.588,66.876,-55.437,180.000,7.544,149.420
C06031=1114.584,67.125,-55.455,-179.998,7.548,149.421
C06032=1114.579,67.374,-55.472,-179.997,7.552,149.421
C06033=1114.574,67.624,-55.490,-179.996,7.556,149.422
C06034=1114.569,67.873,-55.506,-179.994,7.560,149.422
C06035=1114.564,68.122,-55.524,-179.993,7.564,149.423
C06036=1114.558,68.371,-55.541,-179.992,7.569,149.423
C06037=1114.554,68.620,-55.559,-179.990,7.572,149.424
C06038=1114.549,68.870,-55.576,-179.988,7.576,149.424
C06039=1114.544,69.119,-55.594,-179.988,7.580,149.425
C06040=1114.539,69.369,-55.611,-179.986,7.584,149.425
C06041=1114.535,69.618,-55.629,-179.985,7.588,149.426
C06042=1114.529,69.868,-55.646,-179.984,7.592,149.426
C06043=1114.525,70.117,-55.664,-179.982,7.596,149.427
C06044=1114.520,70.366,-55.682,-179.980,7.600,149.427
C06045=1114.515,70.616,-55.698,-179.979,7.604,149.428
C06046=1114.510,70.865,-55.716,-179.978,7.608,149.428
C06047=1114.505,71.114,-55.734,-179.976,7.612,149.429
C06048=1114.500,71.364,-55.752,-179.975,7.616,149.429
C06049=1114.495,71.613,-55.770,-179.974,7.620,149.430
C06050=1114.491,71.862,-55.786,-179.973,7.623,149.430
C06051=1114.486,72.111,-55.804,-179.971,7.627,149.431
C06052=1114.481,72.361,-55.822,-179.970,7.631,149.431
C06053=1114.476,72.610,-55.840,-179.968,7.635,149.432
C06054=1114.471,72.860,-55.858,-179.967,7.639,149.432
C06055=1114.466,73.109,-55.876,-179.966,7.643,149.433
C06056=1114.461,73.358,-55.894,-179.964,7.647,149.433
C06057=1114.456,73.607,-55.910,-179.962,7.651,149.434
C06058=1114.452,73.857,-55.928,-179.961,7.655,149.434
C06059=1114.447,74.106,-55.946,-179.960,7.659,149.435
C06060=1114.442,74.355,-55.964,-179.958,7.663,149.435
C06061=1114.437,74.605,-55.981,-179.957,7.667,149.436
C06062=1114.432,74.854,-55.999,-179.955,7.671,149.436
C06063=1114.427,75.104,-56.018,-179.955,7.675,149.437
C06064=1114.422,75.353,-56.036,-179.953,7.679,149.437
C06065=1114.417,75.602,-56.054,-179.951,7.682,149.438
C06066=1114.412,75.852,-56.071,-179.950,7.687,149.438
C06067=1114.408,76.101,-56.088,-179.949,7.691,149.439
C06068=1114.403,76.350,-56.106,-179.947,7.694,149.439
C06069=1114.398,76.599,-56.124,-179.946,7.698,149.440
C06070=1114.393,76.848,-56.142,-179.944,7.703,149.440
C06071=1114.389,77.063,-56.158,-179.943,7.706,149.441
C06072=1114.385,77.277,-56.173,-179.942,7.709,149.441
C06073=1114.381,77.491,-56.189,-179.942,7.712,149.442
C06074=1114.376,77.705,-56.204,-179.941,7.715,149.442
C06075=1114.372,77.919,-56.220,-179.940,7.719,149.443
C06076=1114.368,78.134,-56.235,-179.939,7.722,149.443
C06077=1114.363,78.348,-56.250,-179.938,7.725,149.444
C06078=1114.360,78.562,-56.266,-179.937,7.728,149.444
C06079=1114.355,78.811,-56.284,-179.937,7.731,149.445
C06080=1114.350,79.060,-56.302,-179.935,7.735,149.445
C06081=1114.345,79.309,-56.320,-179.935,7.739,149.446
C06082=1114.340,79.559,-56.338,-179.933,7.743,149.446
C06083=1114.335,79.808,-56.356,-179.933,7.746,149.447
C06084=1114.331,80.058,-56.375,-179.931,7.751,149.447
C06085=1114.326,80.307,-56.393,-179.930,7.754,149.448
C06086=1114.321,80.556,-56.411,-179.929,7.758,149.448
C06087=1114.316,80.805,-56.429,-179.928,7.761,149.449
C06088=1114.311,81.055,-56.447,-179.927,7.765,149.450
C06089=1114.306,81.304,-56.465,-179.926,7.768,149.450
C06090=1114.302,81.554,-56.483,-179.925,7.773,149.451
C06091=1114.297,81.803,-56.501,-179.924,7.777,149.451
C06092=1114.292,82.052,-56.519,-179.923,7.780,149.452
C06093=1114.287,82.301,-56.537,-179.921,7.784,149.452
C06094=1114.281,82.551,-56.555,-179.921,7.788,149.453
C06095=1114.277,82.801,-56.574,-179.919,7.791,149.453
C06096=1114.272,83.049,-56.592,-179.918,7.796,149.454
C06097=1114.267,83.298,-56.610,-179.917,7.799,149.454
C06098=1114.263,83.547,-56.628,-179.916,7.803,149.455
C06099=1114.258,83.797,-56.646,-179.915,7.806,149.455
C06100=1114.253,84.047,-56.665,-179.914,7.810,149.456
C06101=1114.248,84.296,-56.683,-179.912,7.814,149.456
C06102=1114.243,84.545,-56.701,-179.911,7.817,149.457
C06103=1114.238,84.794,-56.720,-179.910,7.822,149.458
C06104=1114.234,85.044,-56.738,-179.909,7.826,149.458
C06105=1114.229,85.293,-56.756,-179.908,7.829,149.458
C06106=1114.224,85.542,-56.774,-179.907,7.833,149.459
C06107=1114.218,85.791,-56.793,-179.905,7.837,149.459
C06108=1114.214,86.041,-56.812,-179.905,7.840,149.460
C06109=1114.209,86.290,-56.830,-179.903,7.844,149.461
C06110=1114.205,86.539,-56.848,-179.901,7.848,149.461
C06111=1114.199,86.789,-56.866,-179.901,7.852,149.462
C06112=1114.195,87.038,-56.886,-179.899,7.856,149.462
C06113=1114.190,87.287,-56.903,-179.898,7.859,149.463
C06114=1114.185,87.536,-56.921,-179.897,7.864,149.463
C06115=1114.180,87.786,-56.941,-179.896,7.867,149.464
C06116=1114.175,88.035,-56.959,-179.894,7.871,149.464
C06117=1114.171,88.284,-56.977,-179.893,7.875,149.465
C06118=1114.166,88.533,-56.996,-179.891,7.879,149.465
C06119=1114.161,88.783,-57.015,-179.890,7.882,149.466
C06120=1114.156,89.032,-57.033,-179.889,7.886,149.466
C06121=1114.151,89.281,-57.051,-179.888,7.890,149.467
C06122=1114.146,89.531,-57.070,-179.886,7.894,149.467
C06123=1114.141,89.780,-57.088,-179.885,7.897,149.467
C06124=1114.137,90.028,-57.107,-179.884,7.902,149.468
C06125=1114.132,90.278,-57.125,-179.882,7.905,149.469
C06126=1114.127,90.527,-57.145,-179.881,7.909,149.469
C06127=1114.123,90.741,-57.161,-179.880,7.912,149.469
C06128=1114.119,90.956,-57.176,-179.879,7.916,149.470
C06129=1114.115,91.169,-57.192,-179.877,7.919,149.470
C06130=1114.111,91.384,-57.208,-179.876,7.923,149.471
C06131=1114.106,91.598,-57.225,-179.875,7.926,149.471
C06132=1114.103,91.812,-57.241,-179.874,7.928,149.471
C06133=1114.098,92.025,-57.256,-179.872,7.932,149.472
C06134=1114.094,92.240,-57.273,-179.871,7.935,149.472
C06135=1114.089,92.489,-57.291,-179.870,7.939,149.473
C06136=1114.085,92.738,-57.310,-179.868,7.943,149.473
C06137=1114.080,92.987,-57.328,-179.867,7.947,149.474
C06138=1114.075,93.237,-57.348,-179.866,7.951,149.474
C06139=1114.070,93.486,-57.366,-179.864,7.954,149.475
C06140=1114.065,93.735,-57.385,-179.863,7.958,149.475
C06141=1114.060,93.985,-57.403,-179.861,7.962,149.475
C06142=1114.055,94.234,-57.423,-179.859,7.966,149.476
C06143=1114.051,94.483,-57.442,-179.858,7.970,149.476
C06144=1114.045,94.733,-57.460,-179.856,7.974,149.477
C06145=1114.041,94.981,-57.479,-179.855,7.978,149.477
C06146=1114.036,95.231,-57.498,-179.854,7.981,149.478
C06147=1114.031,95.480,-57.517,-179.852,7.985,149.478
C06148=1114.026,95.729,-57.536,-179.851,7.989,149.479
C06149=1114.022,95.979,-57.554,-179.849,7.993,149.479
C06150=1114.017,96.228,-57.574,-179.847,7.996,149.479
C06151=1114.012,96.477,-57.593,-179.846,8.000,149.480
C06152=1114.007,96.727,-57.612,-179.844,8.004,149.480
C06153=1114.003,96.975,-57.630,-179.843,8.008,149.481
C06154=1113.998,97.225,-57.650,-179.841,8.012,149.481
C06155=1113.993,97.474,-57.669,-179.839,8.016,149.482
C06156=1113.988,97.724,-57.688,-179.838,8.020,149.482
C06157=1113.984,97.972,-57.706,-179.836,8.024,149.482
C06158=1113.978,98.221,-57.726,-179.834,8.028,149.483
C06159=1113.974,98.470,-57.745,-179.833,8.031,149.483
C06160=1113.969,98.720,-57.763,-179.831,8.035,149.484
C06161=1113.964,98.970,-57.783,-179.829,8.039,149.484
C06162=1113.960,99.219,-57.802,-179.828,8.043,149.484
C06163=1113.954,99.468,-57.821,-179.826,8.047,149.485
C06164=1113.950,99.717,-57.840,-179.825,8.050,149.485
C06165=1113.945,99.966,-57.859,-179.823,8.054,149.486
C06166=1113.940,100.216,-57.879,-179.822,8.057,149.486
C06167=1113.935,100.465,-57.897,-179.820,8.061,149.486
C06168=1113.931,100.714,-57.917,-179.818,8.065,149.487
C06169=1113.925,100.963,-57.936,-179.816,8.069,149.487
C06170=1113.921,101.212,-57.955,-179.814,8.073,149.488
C06171=1113.916,101.461,-57.975,-179.812,8.077,149.488
C06172=1113.911,101.711,-57.994,-179.811,8.081,149.488
C06173=1113.907,101.959,-58.013,-179.809,8.085,149.489
C06174=1113.902,102.209,-58.033,-179.807,8.088,149.489
C06175=1113.897,102.459,-58.052,-179.805,8.092,149.489
C06176=1113.892,102.708,-58.070,-179.804,8.096,149.490
C06177=1113.888,102.957,-58.090,-179.802,8.099,149.490
C06178=1113.882,103.206,-58.109,-179.800,8.103,149.490
C06179=1113.877,103.456,-58.129,-179.799,8.107,149.491
C06180=1113.873,103.705,-58.148,-179.797,8.111,149.491
C06181=1113.868,103.954,-58.167,-179.795,8.115,149.492
C06182=1113.864,104.203,-58.188,-179.793,8.118,149.492
C06183=1113.860,104.417,-58.204,-179.791,8.122,149.492
C06184=1113.855,104.631,-58.220,-179.790,8.125,149.492
C06185=1113.852,104.845,-58.237,-179.788,8.128,149.493
C06186=1113.847,105.059,-58.254,-179.787,8.131,149.493
C06187=1113.844,105.272,-58.271,-179.785,8.135,149.493
C06188=1113.839,105.487,-58.287,-179.783,8.138,149.494
C06189=1113.835,105.701,-58.305,-179.781,8.141,149.494
C06190=1113.830,105.914,-58.320,-179.780,8.144,149.494
C06191=1113.826,106.164,-58.340,-179.778,8.148,149.494
C06192=1113.821,106.413,-58.360,-179.777,8.152,149.495
C06193=1113.816,106.662,-58.379,-179.775,8.155,149.495
C06194=1113.812,106.911,-58.399,-179.772,8.159,149.495
C06195=1113.807,107.160,-58.419,-179.770,8.163,149.496
C06196=1113.802,107.410,-58.438,-179.768,8.167,149.496
C06197=1113.797,107.659,-58.457,-179.767,8.171,149.496
C06198=1113.792,107.908,-58.477,-179.765,8.174,149.497
C06199=1113.788,108.157,-58.498,-179.762,8.178,149.497
C06200=1113.783,108.406,-58.517,-179.760,8.181,149.497
C06201=1113.778,108.656,-58.536,-179.759,8.185,149.497
C06202=1113.773,108.905,-58.556,-179.757,8.188,149.498
C06203=1113.769,109.153,-58.576,-179.754,8.193,149.498
C06204=1113.764,109.403,-58.595,-179.752,8.197,149.498
C06205=1113.759,109.652,-58.615,-179.750,8.200,149.499
C06206=1113.755,109.901,-58.635,-179.748,8.204,149.499
C06207=1113.750,110.150,-58.654,-179.746,8.207,149.499
C06208=1113.745,110.400,-58.674,-179.744,8.211,149.499
C06209=1113.740,110.649,-58.695,-179.742,8.215,149.500
C06210=1113.736,110.898,-58.714,-179.740,8.219,149.500
C06211=1113.730,111.147,-58.733,-179.738,8.222,149.500
C06212=1113.726,111.396,-58.754,-179.736,8.225,149.500
C06213=1113.721,111.646,-58.774,-179.734,8.229,149.501
C06214=1113.717,111.895,-58.794,-179.733,8.232,149.501
C06215=1113.712,112.144,-58.814,-179.731,8.236,149.501
C06216=1113.707,112.393,-58.833,-179.729,8.239,149.502
C06217=1113.702,112.642,-58.853,-179.728,8.243,149.502
C06218=1113.697,112.891,-58.873,-179.726,8.246,149.502
C06219=1113.693,113.140,-58.893,-179.724,8.250,149.502
C06220=1113.688,113.390,-58.913,-179.722,8.253,149.503
C06221=1113.682,113.639,-58.933,-179.720,8.257,149.503
C06222=1113.678,113.888,-58.953,-179.718,8.260,149.503
C06223=1113.673,114.137,-58.974,-179.717,8.263,149.504
C06224=1113.668,114.387,-58.993,-179.715,8.267,149.504
C06225=1113.664,114.636,-59.014,-179.713,8.270,149.504
C06226=1113.659,114.884,-59.033,-179.712,8.274,149.505
C06227=1113.654,115.133,-59.053,-179.710,8.277,149.505
C06228=1113.650,115.382,-59.074,-179.708,8.281,149.505
C06229=1113.645,115.632,-59.093,-179.706,8.284,149.505
C06230=1113.640,115.881,-59.114,-179.705,8.287,149.506
C06231=1113.635,116.131,-59.134,-179.702,8.291,149.506
C06232=1113.631,116.380,-59.154,-179.700,8.294,149.506
C06233=1113.626,116.628,-59.174,-179.699,8.298,149.507
C06234=1113.621,116.878,-59.194,-179.697,8.301,149.507
C06235=1113.617,117.126,-59.214,-179.695,8.304,149.507
C06236=1113.611,117.376,-59.235,-179.693,8.308,149.507
C06237=1113.607,117.625,-59.255,-179.692,8.312,149.508
C06238=1113.602,117.874,-59.275,-179.690,8.314,149.508
C06239=1113.598,118.088,-59.293,-179.688,8.318,149.508
C06240=1113.594,118.302,-59.310,-179.687,8.321,149.508
C06241=1113.589,118.516,-59.327,-179.685,8.323,149.509
C06242=1113.586,118.730,-59.345,-179.684,8.326,149.509
C06243=1113.582,118.944,-59.362,-179.682,8.329,149.509
C06244=1113.578,119.157,-59.379,-179.680,8.332,149.509
C06245=1113.574,119.371,-59.397,-179.679,8.335,149.510
C06246=1113.569,119.585,-59.414,-179.678,8.338,149.510
C06247=1113.565,119.834,-59.435,-179.676,8.342,149.510
C06248=1113.560,120.083,-59.456,-179.674,8.344,149.510
C06249=1113.555,120.333,-59.475,-179.672,8.348,149.511
C06250=1113.551,120.582,-59.496,-179.671,8.352,149.511
C06251=1113.546,120.831,-59.516,-179.669,8.355,149.511
C06252=1113.541,121.080,-59.537,-179.667,8.358,149.512
C06253=1113.537,121.329,-59.557,-179.665,8.361,149.512
C06254=1113.532,121.578,-59.577,-179.663,8.365,149.512
C06255=1113.527,121.828,-59.598,-179.662,8.368,149.512
C06256=1113.522,122.077,-59.618,-179.660,8.371,149.513
C06257=1113.518,122.326,-59.639,-179.658,8.375,149.513
C06258=1113.513,122.574,-59.659,-179.656,8.378,149.513
C06259=1113.508,122.824,-59.680,-179.655,8.382,149.514
C06260=1113.504,123.073,-59.700,-179.653,8.385,149.514
C06261=1113.499,123.322,-59.721,-179.651,8.389,149.514
C06262=1113.494,123.571,-59.742,-179.649,8.391,149.514
C06263=1113.490,123.820,-59.762,-179.648,8.395,149.515
C06264=1113.485,124.069,-59.783,-179.646,8.399,149.515
C06265=1113.480,124.318,-59.804,-179.644,8.401,149.515
C06266=1113.476,124.567,-59.824,-179.642,8.405,149.515
C06267=1113.471,124.816,-59.845,-179.640,8.409,149.516
C06268=1113.466,125.065,-59.865,-179.638,8.412,149.516
C06269=1113.461,125.314,-59.886,-179.637,8.415,149.516
C06270=1113.456,125.563,-59.907,-179.635,8.418,149.516
C06271=1113.452,125.812,-59.927,-179.633,8.422,149.517
C06272=1113.447,126.062,-59.948,-179.632,8.425,149.517
C06273=1113.442,126.311,-59.968,-179.630,8.429,149.517
C06274=1113.438,126.561,-59.990,-179.628,8.432,149.518
C06275=1113.433,126.810,-60.010,-179.626,8.435,149.518
C06276=1113.428,127.059,-60.031,-179.625,8.439,149.518
C06277=1113.424,127.308,-60.051,-179.623,8.442,149.518
C06278=1113.419,127.557,-60.072,-179.621,8.445,149.519
C06279=1113.414,127.806,-60.093,-179.619,8.448,149.519
C06280=1113.409,128.055,-60.114,-179.617,8.452,149.519
C06281=1113.405,128.304,-60.135,-179.616,8.455,149.520
C06282=1113.400,128.553,-60.156,-179.614,8.458,149.520
C06283=1113.395,128.802,-60.176,-179.612,8.462,149.520
C06284=1113.390,129.051,-60.197,-179.611,8.465,149.520
C06285=1113.386,129.301,-60.218,-179.609,8.468,149.521
C06286=1113.381,129.549,-60.239,-179.607,8.472,149.521
C06287=1113.377,129.798,-60.260,-179.605,8.475,149.521
C06288=1113.372,130.047,-60.281,-179.604,8.479,149.522
C06289=1113.367,130.297,-60.302,-179.602,8.482,149.522
C06290=1113.362,130.546,-60.322,-179.600,8.485,149.522
C06291=1113.357,130.794,-60.344,-179.599,8.489,149.522
C06292=1113.353,131.043,-60.364,-179.596,8.492,149.523
C06293=1113.348,131.293,-60.385,-179.595,8.495,149.523
C06294=1113.343,131.542,-60.407,-179.593,8.498,149.523
C06295=1113.339,131.756,-60.425,-179.591,8.501,149.523
C06296=1113.335,131.969,-60.443,-179.590,8.504,149.524
C06297=1113.332,132.183,-60.460,-179.589,8.507,149.524
C06298=1113.328,132.396,-60.479,-179.587,8.510,149.524
C06299=1113.323,132.611,-60.497,-179.586,8.513,149.525
C06300=1113.319,132.824,-60.515,-179.584,8.516,149.525
C06301=1113.315,133.038,-60.533,-179.583,8.519,149.525
C06302=1113.312,133.252,-60.551,-179.581,8.521,149.525
C06303=1113.307,133.501,-60.572,-179.579,8.525,149.525
C06304=1113.302,133.750,-60.594,-179.578,8.528,149.526
C06305=1113.297,133.999,-60.614,-179.576,8.531,149.526
C06306=1113.292,134.248,-60.636,-179.574,8.535,149.526
C06307=1113.288,134.498,-60.657,-179.573,8.538,149.527
C06308=1113.283,134.747,-60.677,-179.571,8.541,149.527
C06309=1113.278,134.995,-60.699,-179.569,8.545,149.527
C06310=1113.273,135.244,-60.720,-179.568,8.548,149.528
C06311=1113.269,135.494,-60.742,-179.566,8.551,149.528
C06312=1113.265,135.743,-60.762,-179.564,8.555,149.528
C06313=1113.260,135.991,-60.784,-179.563,8.558,149.529
C06314=1113.255,136.241,-60.805,-179.561,8.562,149.529
C06315=1113.251,136.490,-60.827,-179.559,8.565,149.529
C06316=1113.246,136.739,-60.848,-179.558,8.568,149.529
C06317=1113.241,136.988,-60.869,-179.555,8.572,149.530
C06318=1113.236,137.237,-60.890,-179.553,8.575,149.530
C06319=1113.232,137.486,-60.912,-179.552,8.578,149.530
C06320=1113.227,137.735,-60.933,-179.550,8.582,149.531
C06321=1113.222,137.984,-60.954,-179.548,8.585,149.531
C06322=1113.218,138.233,-60.976,-179.547,8.588,149.531
C06323=1113.213,138.482,-60.997,-179.545,8.592,149.531
C06324=1113.208,138.731,-61.019,-179.543,8.595,149.532
C06325=1113.203,138.980,-61.039,-179.542,8.598,149.532
C06326=1113.199,139.229,-61.061,-179.540,8.602,149.532
C06327=1113.194,139.478,-61.083,-179.538,8.606,149.533
C06328=1113.189,139.727,-61.104,-179.537,8.608,149.533
C06329=1113.185,139.976,-61.126,-179.535,8.612,149.533
C06330=1113.180,140.225,-61.148,-179.533,8.616,149.534
C06331=1113.176,140.474,-61.168,-179.532,8.619,149.534
C06332=1113.171,140.723,-61.190,-179.530,8.622,149.534
C06333=1113.166,140.972,-61.212,-179.528,8.626,149.535
C06334=1113.161,141.221,-61.233,-179.527,8.629,149.535
C06335=1113.157,141.471,-61.255,-179.525,8.632,149.535
C06336=1113.152,141.719,-61.277,-179.523,8.636,149.536
C06337=1113.148,141.969,-61.299,-179.522,8.639,149.536
C06338=1113.143,142.218,-61.320,-179.520,8.643,149.536
C06339=1113.138,142.467,-61.341,-179.518,8.646,149.537
C06340=1113.134,142.716,-61.363,-179.517,8.649,149.537
C06341=1113.129,142.964,-61.384,-179.515,8.653,149.537
C06342=1113.125,143.213,-61.406,-179.513,8.656,149.538
C06343=1113.120,143.463,-61.427,-179.512,8.660,149.538
C06344=1113.115,143.711,-61.449,-179.510,8.663,149.538
C06345=1113.111,143.961,-61.471,-179.508,8.667,149.539
C06346=1113.106,144.209,-61.493,-179.507,8.670,149.539
C06347=1113.101,144.458,-61.515,-179.505,8.673,149.539
C06348=1113.097,144.707,-61.537,-179.503,8.677,149.540
C06349=1113.092,144.957,-61.558,-179.502,8.680,149.540
C06350=1113.087,145.206,-61.580,-179.500,8.684,149.540
C06351=1113.083,145.419,-61.598,-179.498,8.687,149.540
C06352=1113.079,145.633,-61.617,-179.496,8.690,149.541
C06353=1113.075,145.846,-61.636,-179.494,8.693,149.541
C06354=1113.072,146.060,-61.655,-179.493,8.696,149.541
C06355=1113.067,146.274,-61.673,-179.491,8.699,149.541
C06356=1113.064,146.487,-61.692,-179.489,8.702,149.542
C06357=1113.060,146.702,-61.711,-179.487,8.706,149.542
C06358=1113.055,146.915,-61.730,-179.486,8.708,149.542
C06359=1113.051,147.164,-61.752,-179.483,8.713,149.542
C06360=1113.046,147.413,-61.774,-179.481,8.716,149.543
C06361=1113.041,147.662,-61.795,-179.479,8.720,149.543
C06362=1113.037,147.911,-61.817,-179.477,8.723,149.543
C06363=1113.032,148.160,-61.839,-179.475,8.727,149.543
C06364=1113.027,148.409,-61.861,-179.473,8.730,149.544
C06365=1113.023,148.658,-61.883,-179.471,8.734,149.544
C06366=1113.018,148.907,-61.905,-179.469,8.737,149.544
C06367=1113.013,149.156,-61.927,-179.467,8.741,149.544
C06368=1113.009,149.405,-61.950,-179.465,8.744,149.545
C06369=1113.004,149.653,-61.971,-179.462,8.749,149.545
C06370=1113.000,149.903,-61.993,-179.460,8.752,149.545
C06371=1112.995,150.151,-62.015,-179.458,8.755,149.545
C06372=1112.990,150.401,-62.037,-179.456,8.759,149.545
C06373=1112.985,150.650,-62.060,-179.453,8.762,149.546
C06374=1112.981,150.899,-62.082,-179.451,8.766,149.546
C06375=1112.977,151.148,-62.104,-179.449,8.769,149.546
C06376=1112.972,151.396,-62.126,-179.447,8.773,149.546
C06377=1112.967,151.646,-62.148,-179.445,8.776,149.547
C06378=1112.962,151.895,-62.170,-179.443,8.780,149.547
C06379=1112.958,152.144,-62.192,-179.441,8.783,149.547
C06380=1112.953,152.392,-62.215,-179.438,8.786,149.547
C06381=1112.949,152.641,-62.237,-179.436,8.790,149.547
C06382=1112.944,152.891,-62.259,-179.434,8.793,149.548
C06383=1112.939,153.140,-62.281,-179.432,8.797,149.548
C06384=1112.935,153.388,-62.304,-179.430,8.800,149.548
C06385=1112.929,153.637,-62.326,-179.428,8.803,149.548
C06386=1112.925,153.887,-62.348,-179.425,8.807,149.548
C06387=1112.921,154.135,-62.371,-179.423,8.810,149.549
C06388=1112.916,154.384,-62.393,-179.421,8.814,149.549
C06389=1112.911,154.634,-62.415,-179.419,8.817,149.549
C06390=1112.907,154.882,-62.438,-179.417,8.820,149.549
C06391=1112.902,155.131,-62.460,-179.415,8.823,149.549
C06392=1112.898,155.380,-62.483,-179.413,8.826,149.549
C06393=1112.893,155.629,-62.505,-179.411,8.830,149.550
C06394=1112.888,155.878,-62.527,-179.409,8.833,149.550
C06395=1112.884,156.127,-62.550,-179.407,8.837,149.550
C06396=1112.879,156.376,-62.572,-179.404,8.840,149.550
C06397=1112.874,156.625,-62.595,-179.402,8.843,149.550
C06398=1112.870,156.874,-62.617,-179.400,8.847,149.551
C06399=1112.865,157.122,-62.640,-179.397,8.850,149.551
C06400=1112.860,157.372,-62.662,-179.395,8.853,149.551
C06401=1112.857,157.620,-62.685,-179.393,8.856,149.551
C06402=1112.851,157.869,-62.707,-179.391,8.859,149.551
C06403=1112.847,158.118,-62.730,-179.389,8.863,149.551
C06404=1112.842,158.368,-62.753,-179.387,8.866,149.551
C06405=1112.838,158.616,-62.776,-179.385,8.869,149.552
C06406=1112.832,158.865,-62.798,-179.382,8.872,149.552
C06407=1112.829,159.079,-62.817,-179.381,8.875,149.552
C06408=1112.826,159.292,-62.837,-179.378,8.878,149.552
C06409=1112.821,159.506,-62.856,-179.377,8.881,149.552
C06410=1112.817,159.719,-62.875,-179.375,8.883,149.552
C06411=1112.813,159.933,-62.895,-179.373,8.887,149.552
C06412=1112.810,160.146,-62.915,-179.371,8.889,149.552
C06413=1112.805,160.361,-62.934,-179.369,8.892,149.553
C06414=1112.801,160.573,-62.953,-179.367,8.894,149.553
C06415=1112.797,160.822,-62.976,-179.365,8.898,149.553
C06416=1112.792,161.072,-62.999,-179.363,8.901,149.553
C06417=1112.788,161.321,-63.022,-179.361,8.904,149.553
C06418=1112.783,161.569,-63.045,-179.358,8.907,149.553
C06419=1112.779,161.818,-63.067,-179.356,8.911,149.553
C06420=1112.774,162.067,-63.090,-179.354,8.913,149.553
C06421=1112.769,162.316,-63.113,-179.352,8.917,149.554
C06422=1112.765,162.565,-63.136,-179.350,8.920,149.554
C06423=1112.760,162.814,-63.158,-179.347,8.923,149.554
C06424=1112.756,163.063,-63.181,-179.345,8.926,149.554
C06425=1112.751,163.312,-63.205,-179.343,8.929,149.554
C06426=1112.747,163.560,-63.227,-179.341,8.932,149.554
C06427=1112.742,163.809,-63.251,-179.338,8.935,149.554
C06428=1112.737,164.058,-63.273,-179.336,8.939,149.555
C06429=1112.733,164.307,-63.296,-179.335,8.941,149.555
C06430=1112.728,164.556,-63.319,-179.332,8.944,149.555
C06431=1112.723,164.805,-63.342,-179.330,8.948,149.555
C06432=1112.719,165.054,-63.365,-179.327,8.951,149.555
C06433=1112.715,165.303,-63.389,-179.325,8.954,149.555
C06434=1112.709,165.551,-63.412,-179.323,8.957,149.555
C06435=1112.705,165.801,-63.434,-179.321,8.960,149.555
C06436=1112.700,166.050,-63.457,-179.319,8.963,149.555
C06437=1112.696,166.299,-63.480,-179.316,8.966,149.556
C06438=1112.692,166.547,-63.503,-179.315,8.969,149.556
C06439=1112.687,166.796,-63.526,-179.312,8.972,149.556
C06440=1112.682,167.045,-63.550,-179.310,8.976,149.556
C06441=1112.678,167.294,-63.573,-179.308,8.979,149.556
C06442=1112.673,167.542,-63.596,-179.306,8.981,149.556
C06443=1112.668,167.792,-63.619,-179.304,8.984,149.556
C06444=1112.664,168.041,-63.642,-179.301,8.988,149.556
C06445=1112.659,168.290,-63.666,-179.299,8.990,149.556
C06446=1112.655,168.538,-63.688,-179.297,8.993,149.557
C06447=1112.650,168.787,-63.712,-179.295,8.997,149.557
C06448=1112.646,169.036,-63.735,-179.292,9.000,149.557
C06449=1112.641,169.285,-63.758,-179.291,9.002,149.557
C06450=1112.636,169.534,-63.782,-179.288,9.005,149.557
C06451=1112.632,169.783,-63.805,-179.286,9.009,149.557
C06452=1112.628,170.032,-63.829,-179.284,9.011,149.557
C06453=1112.623,170.280,-63.852,-179.282,9.014,149.557
C06454=1112.618,170.529,-63.875,-179.279,9.017,149.557
C06455=1112.613,170.778,-63.898,-179.277,9.021,149.558
C06456=1112.608,171.027,-63.922,-179.275,9.023,149.558
C06457=1112.604,171.276,-63.945,-179.273,9.026,149.558
C06458=1112.600,171.525,-63.968,-179.271,9.030,149.558
C06459=1112.595,171.773,-63.992,-179.269,9.032,149.558
C06460=1112.591,172.022,-64.015,-179.266,9.035,149.558
C06461=1112.586,172.271,-64.039,-179.264,9.039,149.558
C06462=1112.581,172.520,-64.062,-179.262,9.041,149.558
C06463=1112.578,172.733,-64.083,-179.260,9.044,149.558
C06464=1112.574,172.947,-64.102,-179.258,9.047,149.559
C06465=1112.570,173.161,-64.123,-179.256,9.049,149.559
C06466=1112.566,173.374,-64.143,-179.254,9.052,149.559
C06467=1112.562,173.587,-64.163,-179.253,9.054,149.559
C06468=1112.559,173.801,-64.183,-179.251,9.057,149.559
C06469=1112.554,174.015,-64.203,-179.249,9.059,149.559
C06470=1112.551,174.228,-64.224,-179.247,9.062,149.559
C06471=1112.546,174.477,-64.247,-179.245,9.065,149.559
C06472=1112.541,174.726,-64.270,-179.243,9.068,149.559
C06473=1112.537,174.974,-64.295,-179.240,9.071,149.559
C06474=1112.532,175.223,-64.318,-179.238,9.073,149.559
C06475=1112.527,175.472,-64.341,-179.236,9.077,149.560
C06476=1112.523,175.720,-64.365,-179.234,9.080,149.560
C06477=1112.518,175.969,-64.389,-179.232,9.082,149.560
C06478=1112.514,176.219,-64.412,-179.230,9.086,149.560
C06479=1112.509,176.467,-64.436,-179.227,9.089,149.560
C06480=1112.504,176.716,-64.460,-179.225,9.091,149.560
C06481=1112.501,176.965,-64.484,-179.223,9.095,149.560
C06482=1112.496,177.214,-64.507,-179.221,9.098,149.560
C06483=1112.492,177.463,-64.531,-179.219,9.100,149.560
C06484=1112.487,177.712,-64.555,-179.217,9.104,149.560
C06485=1112.482,177.960,-64.579,-179.215,9.106,149.561
C06486=1112.478,178.209,-64.602,-179.212,9.109,149.561
C06487=1112.473,178.457,-64.626,-179.210,9.113,149.561
C06488=1112.469,178.706,-64.650,-179.208,9.115,149.561
C06489=1112.464,178.955,-64.674,-179.206,9.118,149.561
C06490=1112.459,179.205,-64.698,-179.204,9.121,149.561
C06491=1112.455,179.453,-64.722,-179.202,9.124,149.561
C06492=1112.450,179.702,-64.745,-179.199,9.127,149.561
C06493=1112.446,179.951,-64.770,-179.197,9.130,149.561
C06494=1112.441,180.200,-64.793,-179.194,9.133,149.561
C06495=1112.437,180.448,-64.817,-179.192,9.136,149.561
C06496=1112.432,180.697,-64.841,-179.189,9.139,149.561
C06497=1112.428,180.946,-64.865,-179.187,9.142,149.561
C06498=1112.423,181.195,-64.889,-179.184,9.146,149.561
C06499=1112.419,181.443,-64.913,-179.182,9.149,149.562
C06500=1112.414,181.693,-64.937,-179.179,9.152,149.562
C06501=1112.410,181.941,-64.961,-179.177,9.155,149.562
C06502=1112.406,182.190,-64.985,-179.175,9.158,149.562
C06503=1112.401,182.439,-65.009,-179.173,9.161,149.562
C06504=1112.396,182.688,-65.033,-179.170,9.164,149.562
C06505=1112.392,182.936,-65.057,-179.167,9.167,149.562
C06506=1112.387,183.185,-65.081,-179.165,9.170,149.562
C06507=1112.383,183.434,-65.105,-179.162,9.173,149.562
C06508=1112.378,183.683,-65.130,-179.160,9.175,149.562
C06509=1112.374,183.931,-65.154,-179.158,9.178,149.562
C06510=1112.369,184.181,-65.177,-179.155,9.181,149.562
C06511=1112.365,184.429,-65.201,-179.153,9.184,149.562
C06512=1112.360,184.678,-65.226,-179.151,9.187,149.562
C06513=1112.356,184.927,-65.251,-179.148,9.190,149.562
C06514=1112.351,185.175,-65.275,-179.146,9.193,149.562
C06515=1112.346,185.424,-65.299,-179.143,9.196,149.562
C06516=1112.342,185.674,-65.323,-179.141,9.198,149.562
C06517=1112.338,185.922,-65.347,-179.139,9.202,149.562
C06518=1112.333,186.171,-65.372,-179.136,9.205,149.562
C06519=1112.329,186.384,-65.392,-179.134,9.207,149.562
C06520=1112.325,186.598,-65.414,-179.132,9.209,149.562
C06521=1112.322,186.811,-65.434,-179.130,9.212,149.562
C06522=1112.318,187.024,-65.455,-179.129,9.214,149.562
C06523=1112.314,187.237,-65.477,-179.127,9.216,149.563
C06524=1112.310,187.451,-65.496,-179.124,9.219,149.563
C06525=1112.306,187.664,-65.517,-179.122,9.222,149.563
C06526=1112.302,187.878,-65.539,-179.120,9.224,149.563
C06527=1112.298,188.126,-65.563,-179.118,9.226,149.563
C06528=1112.292,188.375,-65.588,-179.116,9.230,149.563
C06529=1112.288,188.623,-65.612,-179.113,9.233,149.563
C06530=1112.284,188.873,-65.636,-179.112,9.235,149.563
C06531=1112.279,189.121,-65.661,-179.109,9.238,149.563
C06532=1112.275,189.370,-65.685,-179.107,9.240,149.563
C06533=1112.270,189.619,-65.710,-179.105,9.243,149.563
C06534=1112.266,189.868,-65.734,-179.102,9.247,149.563
C06535=1112.261,190.116,-65.759,-179.100,9.249,149.563
C06536=1112.257,190.365,-65.784,-179.098,9.252,149.563
C06537=1112.252,190.613,-65.809,-179.096,9.254,149.563
C06538=1112.248,190.863,-65.833,-179.093,9.257,149.563
C06539=1112.243,191.111,-65.858,-179.091,9.260,149.563
C06540=1112.239,191.360,-65.882,-179.089,9.263,149.563
C06541=1112.234,191.609,-65.907,-179.086,9.266,149.563
C06542=1112.230,191.858,-65.931,-179.084,9.268,149.563
C06543=1112.225,192.106,-65.955,-179.082,9.271,149.563
C06544=1112.221,192.355,-65.981,-179.080,9.274,149.563
C06545=1112.216,192.603,-66.005,-179.078,9.277,149.564
C06546=1112.212,192.853,-66.030,-179.076,9.280,149.564
C06547=1112.207,193.101,-66.054,-179.074,9.283,149.564
C06548=1112.203,193.350,-66.078,-179.072,9.285,149.564
C06549=1112.199,193.599,-66.104,-179.069,9.288,149.564
C06550=1112.194,193.847,-66.128,-179.067,9.291,149.564
C06551=1112.190,194.096,-66.153,-179.065,9.294,149.564
C06552=1112.184,194.345,-66.178,-179.063,9.296,149.564
C06553=1112.180,194.593,-66.203,-179.061,9.299,149.564
C06554=1112.176,194.842,-66.228,-179.059,9.302,149.564
C06555=1112.171,195.091,-66.252,-179.057,9.305,149.565
C06556=1112.167,195.340,-66.278,-179.055,9.308,149.565
C06557=1112.162,195.588,-66.302,-179.052,9.311,149.565
C06558=1112.158,195.837,-66.327,-179.050,9.313,149.565
C06559=1112.153,196.085,-66.352,-179.049,9.316,149.565
C06560=1112.149,196.335,-66.377,-179.046,9.319,149.565
C06561=1112.145,196.583,-66.401,-179.044,9.322,149.565
C06562=1112.140,196.832,-66.427,-179.041,9.325,149.565
C06563=1112.135,197.081,-66.452,-179.039,9.328,149.565
C06564=1112.131,197.330,-66.476,-179.036,9.331,149.565
C06565=1112.127,197.578,-66.502,-179.034,9.334,149.565
C06566=1112.122,197.827,-66.527,-179.030,9.338,149.565
C06567=1112.118,198.075,-66.551,-179.028,9.341,149.565
C06568=1112.113,198.325,-66.576,-179.025,9.344,149.565
C06569=1112.109,198.573,-66.602,-179.022,9.347,149.565
C06570=1112.105,198.822,-66.626,-179.020,9.350,149.565
C06571=1112.100,199.070,-66.652,-179.017,9.353,149.565
C06572=1112.095,199.319,-66.677,-179.014,9.356,149.565
C06573=1112.091,199.568,-66.702,-179.012,9.359,149.565
C06574=1112.087,199.817,-66.726,-179.009,9.362,149.565
C06575=1112.083,200.029,-66.748,-179.006,9.365,149.565
C06576=1112.079,200.243,-66.770,-179.004,9.367,149.565
C06577=1112.075,200.456,-66.792,-179.001,9.370,149.565
C06578=1112.071,200.669,-66.813,-178.999,9.372,149.565
C06579=1112.068,200.882,-66.835,-178.996,9.375,149.565
C06580=1112.064,201.096,-66.856,-178.995,9.377,149.565
C06581=1112.060,201.309,-66.878,-178.992,9.380,149.565
C06582=1112.056,201.522,-66.899,-178.990,9.382,149.565
C06583=1112.052,201.771,-66.925,-178.987,9.385,149.565
C06584=1112.047,202.020,-66.950,-178.984,9.388,149.564
C06585=1112.043,202.269,-66.975,-178.981,9.391,149.564
C06586=1112.038,202.517,-67.001,-178.978,9.394,149.564
C06587=1112.033,202.766,-67.026,-178.975,9.396,149.564
C06588=1112.030,203.015,-67.051,-178.973,9.400,149.564
C06589=1112.025,203.263,-67.076,-178.970,9.402,149.564
C06590=1112.021,203.512,-67.102,-178.967,9.405,149.564
C06591=1112.016,203.760,-67.127,-178.964,9.408,149.564
C06592=1112.011,204.009,-67.153,-178.961,9.412,149.564
C06593=1112.007,204.258,-67.178,-178.958,9.414,149.564
C06594=1112.002,204.506,-67.204,-178.955,9.417,149.564
C06595=1111.998,204.755,-67.229,-178.952,9.420,149.564
C06596=1111.994,205.004,-67.255,-178.950,9.423,149.564
C06597=1111.989,205.252,-67.280,-178.947,9.426,149.563
C06598=1111.985,205.501,-67.306,-178.944,9.428,149.563
C06599=1111.980,205.750,-67.331,-178.941,9.432,149.563
C06600=1111.975,205.998,-67.357,-178.938,9.434,149.563
C06601=1111.971,206.247,-67.383,-178.935,9.437,149.563
C06602=1111.967,206.496,-67.408,-178.932,9.440,149.563
C06603=1111.962,206.744,-67.434,-178.930,9.443,149.563
C06604=1111.958,206.993,-67.459,-178.927,9.446,149.563
C06605=1111.953,207.242,-67.484,-178.924,9.448,149.563
C06606=1111.949,207.490,-67.510,-178.921,9.451,149.562
C06607=1111.944,207.739,-67.536,-178.918,9.455,149.563
C06608=1111.940,207.988,-67.561,-178.915,9.458,149.562
C06609=1111.936,208.236,-67.587,-178.912,9.461,149.562
C06610=1111.931,208.485,-67.612,-178.909,9.464,149.562
C06611=1111.927,208.733,-67.638,-178.906,9.466,149.562
C06612=1111.923,208.982,-67.664,-178.903,9.469,149.562
C06613=1111.918,209.231,-67.691,-178.901,9.472,149.562
C06614=1111.913,209.479,-67.716,-178.898,9.475,149.562
C06615=1111.909,209.728,-67.742,-178.894,9.478,149.562
C06616=1111.905,209.976,-67.768,-178.892,9.482,149.562
C06617=1111.901,210.225,-67.794,-178.889,9.484,149.562
C06618=1111.896,210.474,-67.819,-178.886,9.487,149.562
C06619=1111.891,210.722,-67.845,-178.883,9.490,149.562
C06620=1111.886,210.971,-67.871,-178.881,9.493,149.562
C06621=1111.883,211.219,-67.898,-178.877,9.497,149.562
C06622=1111.878,211.468,-67.923,-178.875,9.500,149.562
C06623=1111.874,211.717,-67.949,-178.872,9.503,149.562
C06624=1111.869,211.965,-67.975,-178.869,9.506,149.562
C06625=1111.864,212.214,-68.001,-178.866,9.509,149.561
C06626=1111.860,212.462,-68.027,-178.863,9.512,149.562
C06627=1111.856,212.711,-68.053,-178.860,9.515,149.561
C06628=1111.852,212.960,-68.079,-178.858,9.518,149.561
C06629=1111.847,213.209,-68.105,-178.855,9.522,149.562
C06630=1111.842,213.457,-68.131,-178.852,9.525,149.561
C06631=1111.839,213.670,-68.153,-178.850,9.528,149.562
C06632=1111.835,213.884,-68.176,-178.848,9.530,149.562
C06633=1111.831,214.096,-68.198,-178.846,9.532,149.562
C06634=1111.828,214.310,-68.220,-178.844,9.535,149.562
C06635=1111.824,214.523,-68.243,-178.842,9.538,149.562
C06636=1111.820,214.735,-68.266,-178.840,9.540,149.562
C06637=1111.816,214.949,-68.288,-178.839,9.543,149.562
C06638=1111.812,215.161,-68.310,-178.837,9.545,149.562
C06639=1111.808,215.410,-68.336,-178.834,9.548,149.562
C06640=1111.803,215.659,-68.363,-178.833,9.551,149.563
C06641=1111.799,215.908,-68.389,-178.830,9.554,149.563
C06642=1111.795,216.156,-68.415,-178.828,9.557,149.563
C06643=1111.790,216.405,-68.442,-178.825,9.560,149.563
C06644=1111.786,216.653,-68.468,-178.824,9.563,149.563
C06645=1111.782,216.902,-68.494,-178.821,9.566,149.563
C06646=1111.777,217.151,-68.520,-178.819,9.569,149.563
C06647=1111.773,217.399,-68.547,-178.816,9.572,149.563
C06648=1111.769,217.648,-68.572,-178.815,9.575,149.563
C06649=1111.764,217.896,-68.599,-178.812,9.578,149.563
C06650=1111.761,218.145,-68.626,-178.810,9.581,149.564
C06651=1111.756,218.394,-68.652,-178.807,9.584,149.564
C06652=1111.751,218.641,-68.678,-178.805,9.587,149.564
C06653=1111.747,218.890,-68.704,-178.803,9.590,149.564
C06654=1111.742,219.139,-68.731,-178.801,9.593,149.564
C06655=1111.738,219.387,-68.757,-178.798,9.596,149.564
C06656=1111.733,219.636,-68.784,-178.795,9.599,149.564
C06657=1111.729,219.884,-68.810,-178.793,9.603,149.564
C06658=1111.724,220.133,-68.837,-178.791,9.606,149.564
C06659=1111.721,220.381,-68.863,-178.789,9.608,149.565
C06660=1111.716,220.630,-68.890,-178.786,9.611,149.565
C06661=1111.712,220.879,-68.916,-178.784,9.615,149.565
C06662=1111.707,221.127,-68.943,-178.781,9.618,149.565
C06663=1111.703,221.375,-68.970,-178.779,9.621,149.565
C06664=1111.698,221.624,-68.996,-178.776,9.624,149.565
C06665=1111.694,221.873,-69.022,-178.774,9.627,149.565
C06666=1111.690,222.121,-69.049,-178.772,9.630,149.565
C06667=1111.686,222.371,-69.076,-178.769,9.634,149.565
C06668=1111.681,222.619,-69.103,-178.767,9.637,149.565
C06669=1111.677,222.868,-69.130,-178.764,9.640,149.565
C06670=1111.673,223.116,-69.156,-178.762,9.642,149.565
C06671=1111.668,223.364,-69.183,-178.760,9.645,149.566
C06672=1111.664,223.613,-69.209,-178.757,9.648,149.566
C06673=1111.659,223.862,-69.236,-178.755,9.651,149.566
C06674=1111.654,224.110,-69.263,-178.752,9.655,149.566
C06675=1111.651,224.358,-69.290,-178.750,9.658,149.566
C06676=1111.646,224.607,-69.317,-178.747,9.661,149.566
C06677=1111.642,224.855,-69.343,-178.745,9.664,149.566
C06678=1111.637,225.103,-69.370,-178.742,9.667,149.566
C06679=1111.632,225.353,-69.397,-178.739,9.670,149.566
C06680=1111.628,225.601,-69.423,-178.737,9.673,149.566
C06681=1111.624,225.850,-69.450,-178.734,9.676,149.566
C06682=1111.620,226.098,-69.477,-178.731,9.679,149.566
C06683=1111.616,226.347,-69.504,-178.729,9.682,149.566
C06684=1111.611,226.595,-69.531,-178.726,9.685,149.566
C06685=1111.606,226.844,-69.558,-178.723,9.688,149.566
C06686=1111.603,227.092,-69.585,-178.721,9.691,149.566
C06687=1111.599,227.305,-69.608,-178.718,9.694,149.566
C06688=1111.595,227.518,-69.632,-178.716,9.696,149.566
C06689=1111.591,227.731,-69.654,-178.714,9.699,149.566
C06690=1111.587,227.944,-69.678,-178.712,9.702,149.566
C06691=1111.584,228.156,-69.700,-178.709,9.705,149.566
C06692=1111.580,228.370,-69.724,-178.707,9.707,149.566
C06693=1111.576,228.583,-69.747,-178.705,9.709,149.566
C06694=1111.572,228.796,-69.770,-178.702,9.712,149.566
C06695=1111.568,229.044,-69.797,-178.700,9.715,149.566
C06696=1111.564,229.293,-69.824,-178.697,9.718,149.566
C06697=1111.559,229.541,-69.851,-178.694,9.721,149.566
C06698=1111.555,229.790,-69.879,-178.691,9.724,149.566
C06699=1111.551,230.038,-69.906,-178.689,9.727,149.566
C06700=1111.547,230.287,-69.932,-178.686,9.729,149.566
C06701=1111.542,230.535,-69.960,-178.683,9.733,149.566
C06702=1111.537,230.784,-69.987,-178.680,9.735,149.566
C06703=1111.534,231.032,-70.015,-178.677,9.738,149.566
C06704=1111.529,231.281,-70.042,-178.675,9.741,149.566
C06705=1111.524,231.529,-70.069,-178.672,9.744,149.566
C06706=1111.520,231.778,-70.096,-178.669,9.747,149.566
C06707=1111.516,232.026,-70.124,-178.666,9.750,149.566
C06708=1111.512,232.274,-70.151,-178.663,9.753,149.565
C06709=1111.507,232.523,-70.178,-178.660,9.755,149.565
C06710=1111.503,232.771,-70.205,-178.657,9.758,149.565
C06711=1111.499,233.020,-70.233,-178.656,9.760,149.565
C06712=1111.494,233.268,-70.260,-178.653,9.763,149.565
C06713=1111.490,233.517,-70.287,-178.650,9.766,149.565
C06714=1111.486,233.766,-70.315,-178.647,9.769,149.565
C06715=1111.481,234.014,-70.342,-178.644,9.772,149.565
C06716=1111.477,234.262,-70.370,-178.641,9.774,149.565
C06717=1111.472,234.510,-70.397,-178.639,9.776,149.565
C06718=1111.468,234.760,-70.424,-178.636,9.779,149.565
C06719=1111.464,235.007,-70.452,-178.633,9.782,149.565
C06720=1111.459,235.256,-70.479,-178.630,9.785,149.565
C06721=1111.455,235.505,-70.507,-178.628,9.788,149.564
C06722=1111.451,235.753,-70.534,-178.625,9.790,149.564
C06723=1111.446,236.001,-70.562,-178.622,9.793,149.564
C06724=1111.442,236.250,-70.590,-178.620,9.796,149.564
C06725=1111.438,236.498,-70.617,-178.617,9.798,149.564
C06726=1111.433,236.746,-70.644,-178.614,9.800,149.564
C06727=1111.430,236.995,-70.673,-178.612,9.803,149.564
C06728=1111.425,237.244,-70.700,-178.609,9.806,149.564
C06729=1111.421,237.491,-70.727,-178.607,9.808,149.564
C06730=1111.416,237.741,-70.755,-178.604,9.811,149.564
C06731=1111.412,237.989,-70.783,-178.601,9.814,149.564
C06732=1111.408,238.238,-70.810,-178.599,9.816,149.563
C06733=1111.404,238.486,-70.838,-178.596,9.818,149.563
C06734=1111.399,238.734,-70.866,-178.593,9.822,149.563
C06735=1111.395,238.983,-70.894,-178.591,9.823,149.563
C06736=1111.390,239.231,-70.921,-178.588,9.826,149.563
C06737=1111.386,239.479,-70.948,-178.585,9.829,149.563
C06738=1111.382,239.728,-70.977,-178.583,9.831,149.563
C06739=1111.377,239.976,-71.004,-178.580,9.834,149.563
C06740=1111.374,240.224,-71.033,-178.577,9.837,149.563
C06741=1111.368,240.473,-71.060,-178.575,9.839,149.563
C06742=1111.365,240.722,-71.088,-178.572,9.842,149.563
C06743=1111.361,240.935,-71.112,-178.570,9.844,149.563
C06744=1111.357,241.147,-71.136,-178.568,9.846,149.563
C06745=1111.354,241.360,-71.160,-178.566,9.848,149.563
C06746=1111.350,241.573,-71.183,-178.564,9.851,149.563
C06747=1111.347,241.786,-71.207,-178.561,9.853,149.562
C06748=1111.342,241.999,-71.231,-178.560,9.855,149.562
C06749=1111.339,242.211,-71.256,-178.557,9.857,149.562
C06750=1111.335,242.424,-71.279,-178.555,9.859,149.562
C06751=1111.331,242.672,-71.307,-178.552,9.862,149.562
C06752=1111.327,242.921,-71.335,-178.550,9.865,149.562
C06753=1111.322,243.169,-71.363,-178.548,9.867,149.562
C06754=1111.318,243.418,-71.391,-178.545,9.870,149.562
C06755=1111.313,243.666,-71.419,-178.543,9.872,149.562
C06756=1111.310,243.915,-71.447,-178.540,9.875,149.562
C06757=1111.304,244.163,-71.475,-178.538,9.877,149.562
C06758=1111.301,244.411,-71.503,-178.535,9.880,149.562
C06759=1111.296,244.659,-71.531,-178.532,9.883,149.562
C06760=1111.292,244.908,-71.560,-178.531,9.885,149.562
C06761=1111.288,245.156,-71.588,-178.528,9.888,149.562
C06762=1111.284,245.405,-71.616,-178.526,9.890,149.562
C06763=1111.279,245.653,-71.644,-178.523,9.894,149.562
C06764=1111.275,245.901,-71.672,-178.521,9.896,149.562
C06765=1111.271,246.149,-71.700,-178.519,9.899,149.562
C06766=1111.266,246.399,-71.728,-178.517,9.901,149.562
C06767=1111.261,246.647,-71.756,-178.514,9.904,149.562
C06768=1111.258,246.895,-71.784,-178.511,9.907,149.562
C06769=1111.254,247.143,-71.813,-178.510,9.910,149.562
C06770=1111.249,247.391,-71.841,-178.507,9.913,149.562
C06771=1111.245,247.640,-71.870,-178.504,9.916,149.563
C06772=1111.240,247.888,-71.898,-178.501,9.919,149.562
C06773=1111.237,248.137,-71.926,-178.497,9.923,149.562
C06774=1111.232,248.385,-71.954,-178.494,9.925,149.562
C06775=1111.228,248.633,-71.982,-178.490,9.929,149.562
C06776=1111.223,248.882,-72.011,-178.487,9.932,149.562
C06777=1111.219,249.130,-72.039,-178.484,9.935,149.562
C06778=1111.214,249.379,-72.068,-178.481,9.937,149.561
C06779=1111.210,249.626,-72.096,-178.477,9.941,149.561
C06780=1111.206,249.875,-72.125,-178.474,9.944,149.561
C06781=1111.202,250.124,-72.153,-178.471,9.946,149.561
C06782=1111.197,250.372,-72.181,-178.468,9.949,149.561
C06783=1111.193,250.621,-72.209,-178.464,9.952,149.561
C06784=1111.189,250.869,-72.239,-178.461,9.955,149.560
C06785=1111.185,251.117,-72.267,-178.458,9.958,149.560
C06786=1111.180,251.366,-72.295,-178.456,9.960,149.560
C06787=1111.177,251.614,-72.324,-178.452,9.962,149.560
C06788=1111.172,251.862,-72.353,-178.449,9.965,149.560
C06789=1111.168,252.110,-72.381,-178.446,9.967,149.560
C06790=1111.164,252.359,-72.410,-178.443,9.970,149.560
C06791=1111.159,252.607,-72.439,-178.441,9.972,149.559
C06792=1111.155,252.855,-72.467,-178.438,9.975,149.559
C06793=1111.150,253.104,-72.496,-178.435,9.977,149.559
C06794=1111.146,253.352,-72.524,-178.432,9.979,149.559
C06795=1111.142,253.600,-72.553,-178.430,9.981,149.559
C06796=1111.138,253.849,-72.582,-178.427,9.984,149.559
C06797=1111.133,254.097,-72.610,-178.425,9.986,149.558
C06798=1111.129,254.345,-72.639,-178.423,9.988,149.558
C06799=1111.126,254.557,-72.664,-178.421,9.990,149.558
C06800=1111.122,254.771,-72.689,-178.418,9.992,149.558
C06801=1111.119,254.983,-72.713,-178.416,9.995,149.558
C06802=1111.115,255.196,-72.738,-178.415,9.996,149.558
C06803=1111.111,255.408,-72.762,-178.413,9.998,149.558
C06804=1111.108,255.622,-72.787,-178.411,10.000,149.558
C06805=1111.104,255.834,-72.812,-178.409,10.002,149.558
C06806=1111.100,256.047,-72.836,-178.407,10.004,149.558
C06807=1111.096,256.296,-72.865,-178.404,10.007,149.558
C06808=1111.092,256.543,-72.894,-178.402,10.010,149.558
C06809=1111.087,256.792,-72.922,-178.399,10.013,149.558
C06810=1111.083,257.040,-72.952,-178.397,10.015,149.558
C06811=1111.078,257.289,-72.980,-178.394,10.017,149.558
C06812=1111.075,257.537,-73.009,-178.391,10.021,149.558
C06813=1111.071,257.785,-73.039,-178.388,10.023,149.558
C06814=1111.066,258.033,-73.067,-178.385,10.026,149.558
C06815=1111.062,258.282,-73.097,-178.382,10.029,149.558
C06816=1111.058,258.529,-73.125,-178.380,10.032,149.558
C06817=1111.054,258.778,-73.154,-178.377,10.035,149.558
C06818=1111.049,259.026,-73.183,-178.374,10.037,149.558
C06819=1111.045,259.274,-73.213,-178.371,10.040,149.557
C06820=1111.040,259.523,-73.241,-178.368,10.043,149.557
C06821=1111.037,259.771,-73.270,-178.366,10.045,149.557
C06822=1111.033,260.019,-73.300,-178.363,10.048,149.557
C06823=1111.028,260.268,-73.329,-178.360,10.051,149.557
C06824=1111.023,260.516,-73.358,-178.357,10.054,149.557
C06825=1111.019,260.764,-73.387,-178.354,10.056,149.557
C06826=1111.016,261.012,-73.416,-178.352,10.059,149.557
C06827=1111.011,261.261,-73.445,-178.349,10.062,149.557
C06828=1111.007,261.509,-73.474,-178.346,10.065,149.557
C06829=1111.003,261.757,-73.504,-178.343,10.067,149.557
C06830=1110.999,262.006,-73.533,-178.340,10.070,149.556
C06831=1110.994,262.253,-73.562,-178.337,10.073,149.556
C06832=1110.990,262.501,-73.592,-178.334,10.076,149.556
C06833=1110.985,262.750,-73.620,-178.331,10.078,149.556
C06834=1110.981,262.999,-73.650,-178.328,10.081,149.556
C06835=1110.977,263.247,-73.679,-178.325,10.084,149.556
C06836=1110.973,263.495,-73.709,-178.322,10.086,149.556
C06837=1110.968,263.743,-73.738,-178.319,10.089,149.555
C06838=1110.964,263.992,-73.768,-178.316,10.092,149.555
C06839=1110.960,264.240,-73.797,-178.313,10.095,149.555
C06840=1110.955,264.488,-73.826,-178.310,10.097,149.555
C06841=1110.951,264.736,-73.856,-178.307,10.099,149.555
C06842=1110.947,264.984,-73.885,-178.304,10.102,149.555
C06843=1110.943,265.232,-73.914,-178.301,10.104,149.555
C06844=1110.939,265.481,-73.944,-178.299,10.106,149.555
C06845=1110.934,265.729,-73.973,-178.296,10.109,149.554
C06846=1110.930,265.977,-74.003,-178.293,10.112,149.554
C06847=1110.926,266.225,-74.032,-178.290,10.115,149.554
C06848=1110.922,266.474,-74.062,-178.288,10.117,149.554
C06849=1110.918,266.722,-74.091,-178.285,10.119,149.554
C06850=1110.913,266.970,-74.121,-178.282,10.122,149.554
C06851=1110.909,267.219,-74.150,-178.279,10.125,149.554
C06852=1110.905,267.467,-74.180,-178.277,10.127,149.554
C06853=1110.901,267.715,-74.209,-178.274,10.130,149.554
C06854=1110.897,267.963,-74.239,-178.271,10.132,149.553
C06855=1110.893,268.175,-74.264,-178.269,10.134,149.553
C06856=1110.890,268.388,-74.290,-178.266,10.136,149.553
C06857=1110.886,268.600,-74.315,-178.263,10.139,149.553
C06858=1110.882,268.814,-74.341,-178.261,10.141,149.553
C06859=1110.878,269.026,-74.366,-178.259,10.143,149.553
C06860=1110.875,269.239,-74.392,-178.256,10.145,149.553
C06861=1110.871,269.451,-74.417,-178.254,10.147,149.553
C06862=1110.868,269.664,-74.443,-178.251,10.150,149.553
C06863=1110.863,269.912,-74.472,-178.248,10.153,149.552
C06864=1110.860,270.160,-74.502,-178.246,10.155,149.552
C06865=1110.855,270.408,-74.532,-178.243,10.157,149.552
C06866=1110.851,270.657,-74.561,-178.240,10.160,149.552
C06867=1110.847,270.905,-74.591,-178.237,10.163,149.552
C06868=1110.842,271.153,-74.621,-178.234,10.166,149.552
C06869=1110.838,271.401,-74.651,-178.232,10.168,149.552
C06870=1110.834,271.649,-74.680,-178.229,10.170,149.552
C06871=1110.830,271.897,-74.711,-178.226,10.173,149.552
C06872=1110.825,272.145,-74.741,-178.223,10.176,149.551
C06873=1110.821,272.393,-74.771,-178.220,10.179,149.551
C06874=1110.817,272.641,-74.800,-178.217,10.181,149.551
C06875=1110.814,272.890,-74.830,-178.215,10.183,149.551
C06876=1110.809,273.138,-74.861,-178.212,10.186,149.551
C06877=1110.805,273.387,-74.890,-178.209,10.189,149.551
C06878=1110.801,273.634,-74.920,-178.206,10.191,149.551
C06879=1110.797,273.883,-74.950,-178.203,10.194,149.551
C06880=1110.792,274.130,-74.981,-178.200,10.197,149.550
C06881=1110.788,274.379,-75.010,-178.197,10.200,149.550
C06882=1110.784,274.626,-75.040,-178.194,10.202,149.550
C06883=1110.780,274.876,-75.071,-178.192,10.204,149.550
C06884=1110.776,275.123,-75.101,-178.189,10.207,149.550
C06885=1110.772,275.372,-75.130,-178.186,10.210,149.550
C06886=1110.767,275.620,-75.161,-178.183,10.213,149.550
C06887=1110.763,275.868,-75.191,-178.180,10.215,149.550
C06888=1110.759,276.115,-75.221,-178.177,10.218,149.550
C06889=1110.755,276.364,-75.252,-178.174,10.221,149.549
C06890=1110.751,276.612,-75.281,-178.171,10.223,149.549
C06891=1110.746,276.860,-75.312,-178.168,10.226,149.549
C06892=1110.742,277.109,-75.342,-178.165,10.228,149.549
C06893=1110.738,277.356,-75.372,-178.162,10.231,149.549
C06894=1110.734,277.605,-75.403,-178.159,10.233,149.549
C06895=1110.730,277.853,-75.432,-178.156,10.236,149.549
C06896=1110.725,278.101,-75.463,-178.153,10.239,149.549
C06897=1110.722,278.349,-75.493,-178.150,10.241,149.548
C06898=1110.717,278.597,-75.524,-178.147,10.244,149.548
C06899=1110.713,278.846,-75.554,-178.144,10.247,149.548
C06900=1110.709,279.093,-75.584,-178.141,10.250,149.548
C06901=1110.705,279.341,-75.615,-178.138,10.252,149.548
C06902=1110.700,279.589,-75.645,-178.135,10.255,149.548
C06903=1110.697,279.838,-75.675,-178.133,10.257,149.547
C06904=1110.692,280.086,-75.706,-178.129,10.259,149.547
C06905=1110.688,280.334,-75.736,-178.126,10.262,149.547
C06906=1110.684,280.582,-75.767,-178.123,10.265,149.547
C06907=1110.680,280.830,-75.798,-178.120,10.267,149.547
C06908=1110.676,281.078,-75.828,-178.117,10.270,149.547
C06909=1110.671,281.326,-75.858,-178.114,10.272,149.546
C06910=1110.667,281.574,-75.889,-178.111,10.275,149.546
C06911=1110.664,281.786,-75.915,-178.109,10.277,149.546
C06912=1110.661,281.999,-75.941,-178.106,10.279,149.546
C06913=1110.656,282.212,-75.967,-178.103,10.281,149.546
C06914=1110.653,282.424,-75.994,-178.101,10.283,149.546
C06915=1110.650,282.637,-76.020,-178.098,10.285,149.546
C06916=1110.646,282.850,-76.046,-178.095,10.288,149.545
C06917=1110.642,283.061,-76.072,-178.093,10.290,149.545
C06918=1110.639,283.274,-76.098,-178.090,10.292,149.545
C06919=1110.634,283.522,-76.129,-178.087,10.295,149.545
C06920=1110.630,283.771,-76.160,-178.084,10.297,149.545
C06921=1110.627,284.018,-76.190,-178.081,10.300,149.545
C06922=1110.622,284.266,-76.221,-178.078,10.303,149.544
C06923=1110.618,284.515,-76.252,-178.075,10.305,149.544
C06924=1110.614,284.763,-76.282,-178.072,10.308,149.544
C06925=1110.609,285.010,-76.313,-178.069,10.310,149.544
C06926=1110.605,285.259,-76.344,-178.066,10.312,149.544
C06927=1110.602,285.506,-76.375,-178.063,10.315,149.544
C06928=1110.597,285.754,-76.406,-178.060,10.317,149.543
C06929=1110.593,286.003,-76.437,-178.057,10.320,149.543
C06930=1110.589,286.251,-76.468,-178.054,10.322,149.543
C06931=1110.585,286.499,-76.498,-178.051,10.325,149.543
C06932=1110.581,286.747,-76.529,-178.047,10.328,149.543
C06933=1110.576,286.995,-76.560,-178.044,10.330,149.542
C06934=1110.572,287.243,-76.592,-178.042,10.332,149.542
C06935=1110.569,287.491,-76.622,-178.039,10.335,149.542
C06936=1110.565,287.739,-76.653,-178.036,10.338,149.542
C06937=1110.560,287.987,-76.684,-178.033,10.340,149.542
C06938=1110.556,288.235,-76.715,-178.030,10.343,149.542
C06939=1110.552,288.483,-76.746,-178.026,10.345,149.541
C06940=1110.548,288.731,-76.777,-178.023,10.348,149.541
C06941=1110.544,288.980,-76.808,-178.020,10.351,149.541
C06942=1110.539,289.227,-76.839,-178.017,10.353,149.541
C06943=1110.535,289.476,-76.870,-178.015,10.355,149.541
C06944=1110.531,289.724,-76.901,-178.011,10.358,149.541
C06945=1110.527,289.972,-76.933,-178.009,10.360,149.540
C06946=1110.522,290.220,-76.964,-178.005,10.363,149.540
C06947=1110.519,290.467,-76.995,-178.002,10.366,149.540
C06948=1110.515,290.715,-77.026,-177.999,10.368,149.540
C06949=1110.511,290.964,-77.057,-177.996,10.371,149.540
C06950=1110.507,291.211,-77.088,-177.993,10.373,149.540
C06951=1110.503,291.460,-77.119,-177.990,10.375,149.539
C06952=1110.498,291.707,-77.151,-177.987,10.378,149.539
C06953=1110.494,291.956,-77.182,-177.984,10.380,149.539
C06954=1110.490,292.203,-77.214,-177.981,10.383,149.539
C06955=1110.486,292.452,-77.245,-177.978,10.386,149.539
C06956=1110.482,292.699,-77.276,-177.975,10.388,149.539
C06957=1110.478,292.948,-77.307,-177.972,10.391,149.538
C06958=1110.473,293.195,-77.339,-177.969,10.393,149.538
C06959=1110.469,293.444,-77.370,-177.965,10.396,149.538
C06960=1110.465,293.691,-77.401,-177.963,10.398,149.538
C06961=1110.461,293.940,-77.433,-177.960,10.400,149.538
C06962=1110.457,294.188,-77.464,-177.957,10.403,149.537
C06963=1110.453,294.435,-77.496,-177.954,10.406,149.537
C06964=1110.449,294.684,-77.527,-177.950,10.408,149.537
C06965=1110.445,294.931,-77.558,-177.947,10.411,149.537
C06966=1110.441,295.179,-77.590,-177.944,10.413,149.537
C06967=1110.438,295.391,-77.617,-177.942,10.415,149.537
C06968=1110.434,295.604,-77.644,-177.940,10.417,149.537
C06969=1110.431,295.816,-77.671,-177.936,10.420,149.536
C06970=1110.428,296.029,-77.698,-177.934,10.422,149.536
C06971=1110.423,296.240,-77.725,-177.932,10.424,149.536
C06972=1110.420,296.453,-77.752,-177.929,10.427,149.536
C06973=1110.417,296.665,-77.779,-177.926,10.428,149.536
C06974=1110.413,296.877,-77.806,-177.924,10.430,149.536
C06975=1110.409,297.126,-77.837,-177.921,10.433,149.535
C06976=1110.405,297.373,-77.868,-177.917,10.435,149.535
C06977=1110.400,297.622,-77.901,-177.914,10.438,149.535
C06978=1110.397,297.870,-77.933,-177.911,10.441,149.535
C06979=1110.392,298.117,-77.964,-177.908,10.443,149.535
C06980=1110.388,298.366,-77.995,-177.905,10.446,149.534
C06981=1110.385,298.614,-78.027,-177.902,10.449,149.534
C06982=1110.380,298.861,-78.059,-177.899,10.450,149.534
C06983=1110.376,299.110,-78.091,-177.896,10.453,149.534
C06984=1110.372,299.358,-78.123,-177.893,10.455,149.534
C06985=1110.368,299.605,-78.154,-177.890,10.458,149.534
C06986=1110.364,299.853,-78.186,-177.887,10.461,149.533
C06987=1110.360,300.101,-78.218,-177.884,10.463,149.533
C06988=1110.355,300.349,-78.250,-177.880,10.466,149.533
C06989=1110.352,300.597,-78.282,-177.878,10.469,149.533
C06990=1110.348,300.845,-78.314,-177.874,10.471,149.533
C06991=1110.343,301.093,-78.345,-177.872,10.473,149.533
C06992=1110.339,301.341,-78.377,-177.869,10.476,149.532
C06993=1110.335,301.589,-78.409,-177.866,10.478,149.532
C06994=1110.332,301.837,-78.441,-177.862,10.481,149.532
C06995=1110.327,302.084,-78.474,-177.859,10.483,149.532
C06996=1110.323,302.332,-78.505,-177.856,10.486,149.532
C06997=1110.319,302.580,-78.537,-177.853,10.489,149.532
C06998=1110.314,302.828,-78.569,-177.850,10.491,149.531
C06999=1110.310,303.076,-78.601,-177.847,10.494,149.531
C07000=1110.307,303.324,-78.633,-177.844,10.496,149.531
C07001=1110.302,303.572,-78.665,-177.841,10.498,149.531
C07002=1110.298,303.820,-78.697,-177.838,10.501,149.531
C07003=1110.294,304.068,-78.729,-177.835,10.504,149.531
C07004=1110.290,304.316,-78.761,-177.832,10.506,149.530
C07005=1110.286,304.564,-78.794,-177.829,10.509,149.530
C07006=1110.281,304.811,-78.826,-177.825,10.511,149.530
C07007=1110.278,305.059,-78.858,-177.822,10.514,149.530
C07008=1110.274,305.307,-78.890,-177.819,10.516,149.530
C07009=1110.270,305.556,-78.922,-177.816,10.519,149.530
C07010=1110.266,305.803,-78.955,-177.813,10.521,149.529
C07011=1110.261,306.051,-78.987,-177.811,10.524,149.529
C07012=1110.257,306.299,-79.018,-177.807,10.526,149.529
C07013=1110.253,306.546,-79.052,-177.804,10.528,149.529
C07014=1110.250,306.794,-79.083,-177.801,10.531,149.529
C07015=1110.245,307.043,-79.116,-177.798,10.534,149.528
C07016=1110.241,307.291,-79.148,-177.795,10.536,149.528
C07017=1110.237,307.538,-79.181,-177.791,10.539,149.528
C07018=1110.233,307.786,-79.212,-177.788,10.542,149.528
C07019=1110.229,308.034,-79.246,-177.786,10.543,149.528
C07020=1110.225,308.282,-79.277,-177.783,10.546,149.528
C07021=1110.221,308.530,-79.310,-177.779,10.548,149.527
C07022=1110.217,308.777,-79.342,-177.777,10.551,149.527
C07023=1110.214,308.990,-79.370,-177.774,10.553,149.527
C07024=1110.210,309.202,-79.397,-177.771,10.556,149.527
C07025=1110.207,309.414,-79.425,-177.769,10.558,149.527
C07026=1110.203,309.626,-79.453,-177.766,10.559,149.526
C07027=1110.199,309.838,-79.481,-177.763,10.562,149.526
C07028=1110.196,310.050,-79.509,-177.761,10.564,149.526
C07029=1110.193,310.263,-79.537,-177.758,10.566,149.526
C07030=1110.189,310.475,-79.565,-177.755,10.569,149.526
C07031=1110.186,310.723,-79.597,-177.752,10.571,149.526
C07032=1110.181,310.971,-79.630,-177.749,10.574,149.526
C07033=1110.177,311.218,-79.662,-177.746,10.576,149.525
C07034=1110.173,311.466,-79.694,-177.743,10.578,149.525
C07035=1110.169,311.714,-79.727,-177.740,10.581,149.525
C07036=1110.165,311.961,-79.760,-177.737,10.583,149.525
C07037=1110.161,312.210,-79.792,-177.734,10.586,149.525
C07038=1110.157,312.457,-79.825,-177.731,10.589,149.525
C07039=1110.153,312.705,-79.859,-177.727,10.591,149.524
C07040=1110.149,312.953,-79.891,-177.724,10.594,149.524
C07041=1110.145,313.201,-79.924,-177.721,10.596,149.524
C07042=1110.141,313.448,-79.957,-177.718,10.599,149.524
C07043=1110.137,313.697,-79.989,-177.715,10.601,149.524
C07044=1110.133,313.944,-80.022,-177.712,10.603,149.523
C07045=1110.129,314.192,-80.055,-177.709,10.606,149.523
C07046=1110.125,314.440,-80.087,-177.706,10.608,149.523
C07047=1110.121,314.688,-80.120,-177.703,10.611,149.523
C07048=1110.117,314.935,-80.153,-177.700,10.614,149.523
C07049=1110.113,315.183,-80.186,-177.696,10.616,149.523
C07050=1110.109,315.431,-80.218,-177.693,10.619,149.522
C07051=1110.105,315.679,-80.251,-177.690,10.621,149.522
C07052=1110.101,315.927,-80.284,-177.687,10.624,149.522
C07053=1110.096,316.174,-80.318,-177.684,10.626,149.522
C07054=1110.093,316.422,-80.350,-177.681,10.628,149.522
C07055=1110.089,316.670,-80.383,-177.678,10.631,149.522
C07056=1110.085,316.917,-80.416,-177.675,10.633,149.521
C07057=1110.080,317.166,-80.449,-177.672,10.636,149.521
C07058=1110.076,317.413,-80.482,-177.669,10.639,149.521
C07059=1110.073,317.662,-80.516,-177.665,10.641,149.521
C07060=1110.069,317.909,-80.548,-177.662,10.644,149.521
C07061=1110.065,318.157,-80.581,-177.659,10.646,149.520
C07062=1110.061,318.405,-80.614,-177.657,10.648,149.520
C07063=1110.057,318.652,-80.648,-177.653,10.651,149.520
C07064=1110.053,318.900,-80.681,-177.650,10.653,149.520
C07065=1110.049,319.148,-80.714,-177.647,10.656,149.520
C07066=1110.044,319.396,-80.747,-177.644,10.658,149.519
C07067=1110.041,319.643,-80.780,-177.641,10.661,149.519
C07068=1110.037,319.891,-80.813,-177.638,10.664,149.519
C07069=1110.033,320.139,-80.846,-177.634,10.666,149.519
C07070=1110.029,320.387,-80.879,-177.631,10.669,149.519
C07071=1110.025,320.635,-80.913,-177.628,10.671,149.519
C07072=1110.021,320.882,-80.947,-177.625,10.673,149.518
C07073=1110.017,321.129,-80.980,-177.622,10.676,149.518
C07074=1110.013,321.377,-81.013,-177.619,10.678,149.518
C07075=1110.009,321.626,-81.046,-177.616,10.681,149.518
C07076=1110.005,321.873,-81.079,-177.613,10.683,149.518
C07077=1110.001,322.121,-81.113,-177.610,10.686,149.517
C07078=1109.997,322.369,-81.146,-177.607,10.689,149.517
C07079=1109.994,322.580,-81.174,-177.604,10.690,149.517
C07080=1109.990,322.793,-81.203,-177.602,10.692,149.517
C07081=1109.987,323.004,-81.232,-177.598,10.695,149.517
C07082=1109.984,323.217,-81.261,-177.596,10.697,149.517
C07083=1109.980,323.429,-81.289,-177.593,10.699,149.517
C07084=1109.977,323.640,-81.318,-177.590,10.701,149.516
C07085=1109.974,323.853,-81.346,-177.588,10.703,149.516
C07086=1109.970,324.065,-81.375,-177.585,10.706,149.516
C07087=1109.966,324.312,-81.409,-177.582,10.708,149.516
C07088=1109.962,324.560,-81.442,-177.579,10.710,149.516
C07089=1109.958,324.808,-81.475,-177.576,10.713,149.516
C07090=1109.954,325.056,-81.509,-177.573,10.715,149.515
C07091=1109.950,325.303,-81.542,-177.570,10.718,149.515
C07092=1109.946,325.551,-81.576,-177.567,10.720,149.515
C07093=1109.943,325.799,-81.610,-177.563,10.723,149.515
C07094=1109.939,326.047,-81.643,-177.560,10.725,149.515
C07095=1109.934,326.294,-81.677,-177.557,10.728,149.515
C07096=1109.930,326.542,-81.711,-177.554,10.730,149.514
C07097=1109.926,326.790,-81.744,-177.551,10.732,149.514
C07098=1109.923,327.037,-81.778,-177.548,10.735,149.514
C07099=1109.919,327.285,-81.811,-177.545,10.737,149.514
C07100=1109.915,327.532,-81.845,-177.542,10.740,149.513
C07101=1109.910,327.781,-81.879,-177.539,10.743,149.513
C07102=1109.907,328.028,-81.913,-177.535,10.745,149.513
C07103=1109.902,328.276,-81.946,-177.532,10.748,149.513
C07104=1109.899,328.523,-81.980,-177.529,10.750,149.513
C07105=1109.895,328.771,-82.014,-177.526,10.753,149.513
C07106=1109.891,329.019,-82.048,-177.523,10.754,149.512
C07107=1109.887,329.266,-82.082,-177.520,10.757,149.512
C07108=1109.883,329.514,-82.115,-177.517,10.760,149.512
C07109=1109.879,329.762,-82.150,-177.513,10.762,149.512
C07110=1109.874,330.009,-82.183,-177.511,10.765,149.512
C07111=1109.871,330.257,-82.217,-177.507,10.767,149.511
C07112=1109.867,330.504,-82.251,-177.504,10.770,149.511
C07113=1109.862,330.752,-82.285,-177.501,10.772,149.511
C07114=1109.859,331.000,-82.319,-177.498,10.775,149.511
C07115=1109.855,331.247,-82.353,-177.494,10.778,149.511
C07116=1109.851,331.496,-82.387,-177.492,10.779,149.510
C07117=1109.847,331.743,-82.421,-177.489,10.782,149.510
C07118=1109.843,331.990,-82.455,-177.485,10.784,149.510
C07119=1109.840,332.238,-82.490,-177.482,10.787,149.510
C07120=1109.835,332.486,-82.523,-177.479,10.790,149.510
C07121=1109.832,332.733,-82.557,-177.476,10.792,149.510
C07122=1109.828,332.981,-82.592,-177.473,10.795,149.509
C07123=1109.824,333.228,-82.625,-177.469,10.797,149.509
C07124=1109.820,333.476,-82.660,-177.466,10.800,149.509
C07125=1109.816,333.724,-82.693,-177.463,10.802,149.509
C07126=1109.812,333.971,-82.727,-177.460,10.804,149.509
C07127=1109.808,334.219,-82.762,-177.457,10.807,149.509
C07128=1109.804,334.467,-82.796,-177.454,10.809,149.508
C07129=1109.800,334.715,-82.831,-177.451,10.812,149.508
C07130=1109.796,334.962,-82.865,-177.447,10.814,149.508
C07131=1109.793,335.210,-82.899,-177.445,10.817,149.508
C07132=1109.788,335.457,-82.933,-177.441,10.819,149.507
C07133=1109.785,335.705,-82.968,-177.438,10.822,149.507
C07134=1109.781,335.952,-83.002,-177.435,10.825,149.507
C07135=1109.777,336.164,-83.032,-177.432,10.826,149.507
C07136=1109.774,336.376,-83.061,-177.430,10.828,149.507
C07137=1109.771,336.588,-83.090,-177.427,10.831,149.507
C07138=1109.767,336.799,-83.119,-177.424,10.833,149.507
C07139=1109.764,337.012,-83.149,-177.422,10.834,149.506
C07140=1109.761,337.224,-83.178,-177.419,10.837,149.506
C07141=1109.757,337.436,-83.208,-177.416,10.839,149.506
C07142=1109.754,337.648,-83.237,-177.414,10.841,149.506
C07143=1109.750,337.895,-83.271,-177.411,10.843,149.506
C07144=1109.746,338.143,-83.306,-177.407,10.846,149.505
C07145=1109.741,338.390,-83.340,-177.404,10.848,149.505
C07146=1109.738,338.638,-83.375,-177.401,10.851,149.505
C07147=1109.734,338.885,-83.410,-177.398,10.853,149.505
C07148=1109.731,339.133,-83.444,-177.394,10.856,149.505
C07149=1109.726,339.380,-83.478,-177.391,10.858,149.504
C07150=1109.722,339.628,-83.513,-177.389,10.860,149.504
C07151=1109.718,339.875,-83.547,-177.385,10.863,149.504
C07152=1109.714,340.124,-83.582,-177.382,10.865,149.504
C07153=1109.710,340.370,-83.617,-177.379,10.868,149.504
C07154=1109.707,340.618,-83.651,-177.376,10.871,149.504
C07155=1109.702,340.866,-83.686,-177.373,10.873,149.503
C07156=1109.698,341.114,-83.721,-177.369,10.875,149.503
C07157=1109.695,341.361,-83.756,-177.366,10.878,149.503
C07158=1109.691,341.608,-83.790,-177.363,10.880,149.503
C07159=1109.687,341.856,-83.825,-177.360,10.883,149.503
C07160=1109.682,342.104,-83.859,-177.357,10.885,149.502
C07161=1109.679,342.351,-83.894,-177.354,10.887,149.502
C07162=1109.675,342.599,-83.929,-177.350,10.890,149.502
C07163=1109.671,342.847,-83.964,-177.347,10.893,149.502
C07164=1109.667,343.094,-83.999,-177.344,10.895,149.502
C07165=1109.663,343.341,-84.033,-177.341,10.897,149.501
C07166=1109.660,343.589,-84.069,-177.338,10.900,149.501
C07167=1109.656,343.837,-84.103,-177.334,10.902,149.501
C07168=1109.651,344.084,-84.138,-177.331,10.905,149.501
C07169=1109.648,344.331,-84.173,-177.329,10.907,149.501
C07170=1109.644,344.579,-84.207,-177.325,10.909,149.500
C07171=1109.640,344.826,-84.243,-177.322,10.912,149.500
C07172=1109.636,345.075,-84.278,-177.319,10.914,149.500
C07173=1109.632,345.321,-84.313,-177.316,10.917,149.500
C07174=1109.629,345.569,-84.347,-177.312,10.919,149.500
C07175=1109.625,345.817,-84.383,-177.309,10.922,149.499
C07176=1109.620,346.064,-84.417,-177.306,10.924,149.499
C07177=1109.617,346.312,-84.453,-177.303,10.927,149.499
C07178=1109.613,346.559,-84.488,-177.300,10.930,149.499
C07179=1109.608,346.806,-84.523,-177.297,10.931,149.499
C07180=1109.605,347.054,-84.558,-177.294,10.934,149.498
C07181=1109.601,347.302,-84.593,-177.290,10.936,149.498
C07182=1109.597,347.549,-84.628,-177.287,10.939,149.498
C07183=1109.594,347.796,-84.663,-177.284,10.941,149.498
C07184=1109.590,348.044,-84.698,-177.281,10.944,149.498
C07185=1109.586,348.292,-84.734,-177.277,10.946,149.497
C07186=1109.582,348.538,-84.769,-177.274,10.949,149.497
C07187=1109.578,348.787,-84.804,-177.271,10.951,149.497
C07188=1109.574,349.034,-84.839,-177.268,10.953,149.497
C07189=1109.570,349.282,-84.875,-177.265,10.955,149.497
C07190=1109.566,349.528,-84.910,-177.262,10.958,149.496
C07191=1109.563,349.741,-84.940,-177.259,10.961,149.496
C07192=1109.560,349.952,-84.970,-177.256,10.962,149.496
C07193=1109.556,350.164,-85.001,-177.254,10.964,149.496
C07194=1109.553,350.376,-85.030,-177.250,10.967,149.496
C07195=1109.550,350.587,-85.060,-177.248,10.969,149.495
C07196=1109.547,350.799,-85.091,-177.245,10.971,149.495
C07197=1109.543,351.011,-85.122,-177.242,10.973,149.495
C07198=1109.540,351.223,-85.151,-177.239,10.976,149.495
C07199=1109.536,351.471,-85.187,-177.235,10.978,149.495
C07200=1109.532,351.718,-85.222,-177.232,10.980,149.494
C07201=1109.528,351.965,-85.257,-177.229,10.983,149.494
C07202=1109.525,352.213,-85.293,-177.226,10.985,149.494
C07203=1109.521,352.460,-85.328,-177.223,10.987,149.494
C07204=1109.517,352.708,-85.364,-177.220,10.990,149.494
C07205=1109.513,352.954,-85.399,-177.216,10.992,149.493
C07206=1109.509,353.202,-85.435,-177.213,10.994,149.493
C07207=1109.505,353.450,-85.471,-177.210,10.997,149.493
C07208=1109.501,353.697,-85.506,-177.206,10.999,149.493
C07209=1109.498,353.945,-85.542,-177.203,11.002,149.492
C07210=1109.494,354.192,-85.578,-177.200,11.004,149.492
C07211=1109.490,354.440,-85.613,-177.196,11.007,149.492
C07212=1109.486,354.686,-85.648,-177.193,11.009,149.492
C07213=1109.482,354.934,-85.684,-177.189,11.011,149.491
C07214=1109.478,355.182,-85.720,-177.186,11.014,149.491
C07215=1109.474,355.429,-85.756,-177.183,11.016,149.491
C07216=1109.471,355.677,-85.791,-177.179,11.019,149.491
C07217=1109.467,355.924,-85.827,-177.176,11.021,149.490
C07218=1109.463,356.172,-85.862,-177.173,11.024,149.490
C07219=1109.460,356.419,-85.898,-177.169,11.026,149.490
C07220=1109.456,356.666,-85.935,-177.166,11.029,149.490
C07221=1109.452,356.914,-85.970,-177.162,11.031,149.489
C07222=1109.448,357.161,-86.005,-177.159,11.033,149.489
C07223=1109.444,357.408,-86.041,-177.156,11.036,149.489
C07224=1109.440,357.655,-86.078,-177.153,11.038,149.489
C07225=1109.436,357.903,-86.113,-177.149,11.041,149.489
C07226=1109.433,358.150,-86.149,-177.146,11.043,149.488
C07227=1109.429,358.398,-86.184,-177.142,11.045,149.488
C07228=1109.425,358.645,-86.221,-177.139,11.048,149.488
C07229=1109.421,358.893,-86.257,-177.136,11.050,149.487
C07230=1109.418,359.140,-86.292,-177.132,11.053,149.487
C07231=1109.414,359.387,-86.329,-177.129,11.055,149.487
C07232=1109.410,359.635,-86.365,-177.126,11.058,149.487
C07233=1109.406,359.882,-86.400,-177.122,11.060,149.486
C07234=1109.403,360.129,-86.437,-177.119,11.062,149.486
C07235=1109.398,360.377,-86.473,-177.116,11.064,149.486
C07236=1109.395,360.624,-86.509,-177.113,11.066,149.486
C07237=1109.391,360.871,-86.544,-177.109,11.069,149.486
C07238=1109.387,361.119,-86.581,-177.106,11.071,149.485
C07239=1109.384,361.366,-86.617,-177.102,11.073,149.485
C07240=1109.380,361.614,-86.652,-177.099,11.076,149.485
C07241=1109.376,361.861,-86.689,-177.096,11.078,149.484
C07242=1109.372,362.108,-86.725,-177.093,11.081,149.484
C07243=1109.368,362.355,-86.762,-177.089,11.083,149.484
C07244=1109.364,362.603,-86.797,-177.086,11.085,149.484
C07245=1109.361,362.850,-86.834,-177.082,11.088,149.483
C07246=1109.357,363.098,-86.870,-177.079,11.090,149.483
C07247=1109.352,363.426,-86.919,-177.075,11.093,149.483
C07248=1109.348,363.753,-86.966,-177.070,11.097,149.483
C07249=1109.343,364.081,-87.014,-177.065,11.100,149.482
C07250=1109.338,364.409,-87.063,-177.061,11.103,149.482
C07251=1109.086,353.425,-85.527,-177.209,10.998,149.493
C07252=1109.090,353.177,-85.491,-177.212,10.995,149.493
C07253=1109.094,352.930,-85.456,-177.216,10.993,149.493
C07254=1109.097,352.682,-85.420,-177.219,10.990,149.494
C07255=1109.101,352.435,-85.385,-177.222,10.988,149.494
C07256=1109.105,352.188,-85.350,-177.226,10.985,149.494
C07257=1109.109,351.940,-85.314,-177.229,10.983,149.494
C07258=1109.113,351.693,-85.279,-177.232,10.980,149.494
C07259=1109.116,351.445,-85.243,-177.235,10.978,149.495
C07260=1109.120,351.206,-85.209,-177.239,10.976,149.495
C07261=1109.124,350.967,-85.175,-177.242,10.973,149.495
C07262=1109.128,350.727,-85.140,-177.245,10.971,149.495
C07263=1109.131,350.487,-85.106,-177.249,10.968,149.496
C07264=1109.136,350.248,-85.072,-177.251,10.966,149.496
C07265=1109.140,350.008,-85.038,-177.254,10.964,149.496
C07266=1109.143,349.769,-85.004,-177.258,10.961,149.496
C07267=1109.146,349.529,-84.970,-177.261,10.959,149.496
C07268=1109.151,349.282,-84.934,-177.264,10.956,149.497
C07269=1109.154,349.035,-84.899,-177.268,10.954,149.497
C07270=1109.158,348.787,-84.863,-177.271,10.951,149.497
C07271=1109.162,348.539,-84.828,-177.274,10.949,149.497
C07272=1109.166,348.293,-84.793,-177.276,10.947,149.497
C07273=1109.170,348.045,-84.758,-177.280,10.944,149.498
C07274=1109.174,347.797,-84.723,-177.283,10.942,149.498
C07275=1109.177,347.550,-84.688,-177.286,10.939,149.498
C07276=1109.181,347.303,-84.653,-177.289,10.937,149.498
C07277=1109.185,347.055,-84.618,-177.293,10.934,149.498
C07278=1109.189,346.808,-84.583,-177.296,10.932,149.498
C07279=1109.193,346.560,-84.548,-177.299,10.929,149.499
C07280=1109.197,346.312,-84.512,-177.303,10.927,149.499
C07281=1109.201,346.065,-84.477,-177.305,10.925,149.499
C07282=1109.205,345.817,-84.442,-177.308,10.922,149.499
C07283=1109.208,345.570,-84.407,-177.311,10.920,149.499
C07284=1109.212,345.322,-84.373,-177.315,10.917,149.500
C07285=1109.216,345.075,-84.337,-177.318,10.915,149.500
C07286=1109.220,344.827,-84.303,-177.321,10.913,149.500
C07287=1109.225,344.580,-84.267,-177.324,10.910,149.500
C07288=1109.229,344.332,-84.233,-177.328,10.907,149.500
C07289=1109.231,344.085,-84.198,-177.331,10.905,149.501
C07290=1109.236,343.838,-84.163,-177.334,10.902,149.501
C07291=1109.240,343.590,-84.128,-177.337,10.901,149.501
C07292=1109.244,343.342,-84.093,-177.340,10.898,149.501
C07293=1109.247,343.095,-84.059,-177.343,10.895,149.501
C07294=1109.251,342.847,-84.023,-177.346,10.893,149.502
C07295=1109.256,342.600,-83.989,-177.350,10.891,149.502
C07296=1109.260,342.352,-83.954,-177.353,10.888,149.502
C07297=1109.263,342.105,-83.919,-177.356,10.885,149.502
C07298=1109.267,341.857,-83.885,-177.359,10.883,149.502
C07299=1109.271,341.609,-83.850,-177.363,10.880,149.503
C07300=1109.276,341.362,-83.815,-177.365,10.879,149.503
C07301=1109.279,341.115,-83.780,-177.368,10.876,149.503
C07302=1109.283,340.867,-83.746,-177.372,10.873,149.503
C07303=1109.287,340.619,-83.711,-177.375,10.871,149.503
C07304=1109.290,340.371,-83.677,-177.378,10.869,149.504
C07305=1109.295,340.124,-83.642,-177.381,10.866,149.504
C07306=1109.299,339.876,-83.607,-177.384,10.863,149.504
C07307=1109.302,339.629,-83.573,-177.388,10.861,149.504
C07308=1109.306,339.381,-83.538,-177.391,10.858,149.504
C07309=1109.310,339.134,-83.504,-177.394,10.856,149.505
C07310=1109.314,338.886,-83.469,-177.397,10.854,149.505
C07311=1109.319,338.639,-83.434,-177.400,10.851,149.505
C07312=1109.322,338.391,-83.400,-177.403,10.849,149.505
C07313=1109.326,338.144,-83.365,-177.407,10.847,149.505
C07314=1109.330,337.896,-83.331,-177.409,10.844,149.505
C07315=1109.334,337.649,-83.297,-177.413,10.841,149.506
C07316=1109.337,337.436,-83.267,-177.415,10.840,149.506
C07317=1109.341,337.225,-83.238,-177.418,10.837,149.506
C07318=1109.344,337.013,-83.208,-177.421,10.835,149.506
C07319=1109.348,336.801,-83.179,-177.423,10.833,149.506
